# B&R Automation Studio project NAELD004C00R10L518F00 (part 39)

#### Local.var
```iecst
(*2021-08-01*)
(**)
(*Local Action, State & Status*)
VAR
	eAct : eHermesAction := HermesActIdle;
	eStat : eHermesAction := HermesActIdle;
	eMainStatus : eFBStatus := Idle;
	eStatus : eFBStatus := Idle;
	eStatus1 : eFBStatus := Idle;
	eStatus2 : eFBStatus := Idle;
	eStatus3 : eFBStatus := Idle;
	udiStatus : UDINT := 0;
	udiStatus1 : UDINT := 0;
	udiStatus2 : UDINT := 0;
	udiStatus3 : UDINT := 0;
	udiStatus4 : UDINT := 0;
	sStatTxt : STRING[200] := '';
	a_sStatText : ARRAY[0..50] OF STRING[200] := ['Idling','Background Starting Operations','Background Stopping Operations','Deleting Old Log File','Creating Directory','Writing Retain File','Reading Retain File','Saving Configuration',43('')];
END_VAR
(**)
(*Local Alarm*)
VAR
	tyAlmData : tyAlmDat;
	tyAlmData1 : tyAlmDat;
	tyAlmData2 : tyAlmDat;
	tyAlmData3 : tyAlmDat;
	tyAlmData4 : tyAlmDat;
	a_tyAlmText : ARRAY[10000..10199] OF tyAlmTxt := [(sAlmText:='Invalid Ident While Creating Server',sRcyText:='Problem Occurred In The TCP/IP Connection. Check The Connection And Try To Reconnect.'),(sAlmText:='Setting Keep Alive Interval Time Error While Creating Server',sRcyText:='Unable To Establish Connection Between Machine. Check For Setting And Resume Operation.'),(sAlmText:='Setting Keep Alive Idle Time Error While Creating Server',sRcyText:='Unable To Establish Connection Between Machine. Check For Setting And Resume Operation.'),(sAlmText:='Setting Keep Alive Count Error While Creating Server',sRcyText:='Unable To Establish Connection Between Machine. Check For Setting And Resume Operation.'),(sAlmText:='Setting Keep Alive Error While Creating Server',sRcyText:='Unable To Establish Connection Between Machine. Check For Setting And Resume Operation.'),(sAlmText:='Setting Receive Buffer Error While Creating Server',sRcyText:='Unable To Establish Connection Between Machine. Check For Setting And Resume Operation.'),(sAlmText:='Setting Send Buffer Error While Creating Server',sRcyText:='Unable To Establish Connection Between Machine. Check For Setting And Resume Operation.'),(sAlmText:='Setting No Waiting Error While Creating Server',sRcyText:='Unable To Establish Connection Between Machine. Check For Setting And Resume Operation.'),(sAlmText:='TCP Open Port Error While Creating Server',sRcyText:='Problem Occurred In The TCP/IP Connection. Check The Connection And Try To Reconnect.'),(sAlmText:='Closing TCP Error While Creating Server',sRcyText:='Problem Occurred In The TCP/IP Connection. Check The Connection And Try To Reconnect.'),(sAlmText:='Invalid Ident While Listening Client',sRcyText:='There Was A Problem Connecting To The Server. The Server May Not Exist or It is Unavailable At This Time. Check The Connection and Try Again.'),0,(sAlmText:='DS Hermes Connection Lost',sRcyText:='There Was A Problem Connecting To The Server. The Server May Not Exist or It is Unavailable At This Time. Check The Connection and Try Again.'),0,(sAlmText:='Invalid Ident While Receiving Data',sRcyText:='Problem Occurred In The TCP/IP Connection. Check The Connection And Try To Reconnect.'),(sAlmText:='TCP Receive Data Error While Receiving Data',sRcyText:='Problem Occurred In The TCP/IP Connection. Check The Connection And Try To Reconnect.'),(sAlmText:='Receive BoardAvailable While Downstream In Not Connected State',sRcyText:='Receive Illegal Message.'),(sAlmText:='Receive RevokeBoardAvailable While Downstream In Not Connected State',sRcyText:='Receive Illegal Message.'),(sAlmText:='Receive MachineReady While Downstream In Not Connected State',sRcyText:='Receive Illegal Message.'),(sAlmText:='Receive RevokeMachineReady While Downstream In Not Connected State',sRcyText:='Receive Illegal Message.'),(sAlmText:='Receive StartTransport While Downstream In Not Connected State',sRcyText:='Receive Illegal Message.'),(sAlmText:='Receive StopTransport While Downstream In Not Connected State',sRcyText:='Receive Illegal Message.'),(sAlmText:='Receive TransportFinished While Downstream In Not Connected State',sRcyText:='Receive Illegal Message.'),(sAlmText:='Receive BoardForecast While Downstream In Not Connected State',sRcyText:='Receive Illegal Message.'),(sAlmText:='Receive ServiceDescription While Downstream In Service Description State',sRcyText:='Receive Illegal Message.'),(sAlmText:='Receive BoardAvailable While Downstream In Service Description State',sRcyText:='Receive Illegal Message.'),(sAlmText:='Receive RevokeBoardAvailable While Downstream In Service Description State',sRcyText:='Receive Illegal Message.'),(sAlmText:='Receive MachineReady While Downstream In Service Description State',sRcyText:='Receive Illegal Message.'),(sAlmText:='Receive RevokeMachineReady While Downstream In Service Description State',sRcyText:='Receive Illegal Message.'),(sAlmText:='Receive StartTransport While Downstream In Service Description State',sRcyText:='Receive Illegal Message.'),(sAlmText:='Receive StopTransport While Downstream In Service Description State',sRcyText:='Receive Illegal Message.'),(sAlmText:='Receive TransportFinished While Downstream In Service Description State',sRcyText:='Receive Illegal Message.'),(sAlmText:='Receive BoardForecast While Downstream In Service Description State',sRcyText:='Receive Illegal Message.'),(sAlmText:='Receive ServiceDescription While Downstream In Not Available Not Ready State',sRcyText:='Receive Illegal Message.'),(sAlmText:='Receive BoardAvailable While Downstream In Not Available Not Ready State',sRcyText:='Receive Illegal Message.'),(sAlmText:='Receive RevokeBoardAvailable While Downstream In Not Available Not Ready State',sRcyText:='Receive Illegal Message.'),(sAlmText:='Receive RevokeMachineReady While Downstream In Not Available Not Ready State',sRcyText:='Receive Illegal Message.'),(sAlmText:='Receive StartTransport While Downstream In Not Available Not Ready State',sRcyText:='Receive Illegal Message.'),(sAlmText:='Receive StopTransport While Downstream In Not Available Not Ready State',sRcyText:='Receive Illegal Message.'),(sAlmText:='Receive TransportFinished While Downstream In Not Available Not Ready State',sRcyText:='Receive Illegal Message.'),(sAlmText:='Receive BoardForecast While Downstream In Not Available Not Ready State',sRcyText:='Receive Illegal Message.'),(sAlmText:='Receive ServiceDescription While Downstream In Board Available State',sRcyText:='Receive Illegal Message.'),(sAlmText:='Receive BoardAvailable While Downstream In Board Available State',sRcyText:='Receive Illegal Message.'),(sAlmText:='Receive RevokeBoardAvailable While Downstream In Board Available State',sRcyText:='Receive Illegal Message.'),(sAlmText:='Receive RevokeMachineReady While Downstream In Board Available State',sRcyText:='Receive Illegal Message.'),(sAlmText:='Receive StartTransport While Downstream In Board Available State',sRcyText:='Receive Illegal Message.'),(sAlmText:='Receive StopTransport While Downstream In Board Available State',sRcyText:='Receive Illegal Message.'),(sAlmText:='Receive TransportFinished While Downstream In Board Available State',sRcyText:='Receive Illegal Message.'),(sAlmText:='Receive BoardForecast While Downstream In Board Available State',sRcyText:='Receive Illegal Message.'),(sAlmText:='Receive ServiceDescription While Downstream In Machine Ready State',sRcyText:='Receive Illegal Message.'),(sAlmText:='Receive BoardAvailable While Downstream In Machine Ready State',sRcyText:='Receive Illegal Message.'),(sAlmText:='Receive RevokeBoardAvailable While Downstream In Machine Ready State',sRcyText:='Receive Illegal Message.'),(sAlmText:='Receive MachineReady While Downstream In Machine Ready State',sRcyText:='Receive Illegal Message.'),(sAlmText:='Receive StopTransport While Downstream In Machine Ready State',sRcyText:='Receive Illegal Message.'),(sAlmText:='Receive TransportFinished While Downstream In Machine Ready State',sRcyText:='Receive Illegal Message.'),(sAlmText:='Receive BoardForecast While Downstream In Machine Ready State',sRcyText:='Receive Illegal Message.'),(sAlmText:='Receive ServiceDescription While Downstream In Available And Ready State',sRcyText:='Receive Illegal Message.'),(sAlmText:='Receive BoardAvailable While Downstream In Available And Ready State',sRcyText:='Receive Illegal Message.'),(sAlmText:='Receive RevokeBoardAvailable While Downstream In Available And Ready State',sRcyText:='Receive Illegal Message.'),(sAlmText:='Receive MachineReady While Downstream In Available And Ready State',sRcyText:='Receive Illegal Message.'),(sAlmText:='Receive StopTransport While Downstream In Available And Ready State',sRcyText:='Receive Illegal Message.'),(sAlmText:='Receive TransportFinished While Downstream In Available And Ready State',sRcyText:='Receive Illegal Message.'),(sAlmText:='Receive BoardForecast While Downstream In Available And Ready State',sRcyText:='Receive Illegal Message.'),(sAlmText:='Receive ServiceDescription While Downstream In Transporting State',sRcyText:='Receive Illegal Message.'),(sAlmText:='Receive BoardAvailable While Downstream In Transporting State',sRcyText:='Receive Illegal Message.'),(sAlmText:='Receive RevokeBoardAvailable While Downstream In Transporting State',sRcyText:='Receive Illegal Message.'),(sAlmText:='Receive MachineReady While Downstream In Transporting State',sRcyText:='Receive Illegal Message.'),(sAlmText:='Receive RevokeMachineReady While Downstream In Transporting State',sRcyText:='Receive Illegal Message.'),(sAlmText:='Receive StartTransport While Downstream In Transporting State',sRcyText:='Receive Illegal Message.'),(sAlmText:='Receive TransportFinished While Downstream In Transporting State',sRcyText:='Receive Illegal Message.'),(sAlmText:='Receive BoardForecast While Downstream In Transporting State',sRcyText:='Receive Illegal Message.'),(sAlmText:='Receive ServiceDescription While In Transport Finished State',sRcyText:='Receive Illegal Message.'),(sAlmText:='Receive BoardAvailable While In Transport Finished State',sRcyText:='Receive Illegal Message.'),(sAlmText:='Receive RevokeBoardAvailable While In Transport Finished State',sRcyText:='Receive Illegal Message.'),(sAlmText:='Receive MachineReady While In Transport Finished State',sRcyText:='Receive Illegal Message.'),(sAlmText:='Receive RevokeMachineReady While In Transport Finished State',sRcyText:='Receive Illegal Message.'),(sAlmText:='Receive StartTransport While In Transport Finished State',sRcyText:='Receive Illegal Message.'),(sAlmText:='Receive TransportFinished While In Transport Finished State',sRcyText:='Receive Illegal Message.'),(sAlmText:='Receive BoardForecast While In Transport Finished State',sRcyText:='Receive Illegal Message.'),(sAlmText:='Receive ServiceDescription While Downstream In Transport Stopped State',sRcyText:='Receive Illegal Message.'),(sAlmText:='Receive BoardAvailable While Downstream In Transport Stopped State',sRcyText:='Receive Illegal Message.'),(sAlmText:='Receive RevokeBoardAvailable While Downstream In Transport Stopped State',sRcyText:='Receive Illegal Message.'),(sAlmText:='Receive MachineReady While Downstream In Transport Stopped State',sRcyText:='Receive Illegal Message.'),(sAlmText:='Receive RevokeMachineReady While Downstream In Transport Stopped State',sRcyText:='Receive Illegal Message.'),(sAlmText:='Receive StartTransport While Downstream In Transport Stopped State',sRcyText:='Receive Illegal Message.'),(sAlmText:='Receive StopTransport While Downstream In Transport Stopped State',sRcyText:='Receive Illegal Message.'),(sAlmText:='LaneId Mismatch While Checking Service Description',sRcyText:='The LaneId Value Does Not Match. Change The Value And Resend The Value.'),(sAlmText:='MachineId Missing While Checking Service Description',sRcyText:='Missing Input Value For MachineId. Fill Up The Value And Resend.'),(sAlmText:='LandId Out Of Range While Checking Service Description',sRcyText:='LaneId Does Not Fall Within The Expected Range.'),(sAlmText:='LandId Missing While Checking Service Description',sRcyText:='Missing Input Value For LaneId. Fill Up The Value And Resend.'),(sAlmText:='Version Missing While Checking Service Description',sRcyText:='Missing Input Value For Version. Fill Up The Value And Resend.'),(sAlmText:='SupportedFeatures Missing While Checking Service Description',sRcyText:='Missing Input Value For SupportedFeatures. Fill Up The Value And Resend.'),(sAlmText:='NotificationCode Out Of Range While Checking Notification',sRcyText:='NotificationCode Does Not Fall Within The Expected Range.'),(sAlmText:='NotificationCode Missing While Checking Notification',sRcyText:='Missing Input Value For NotificationCode. Fill Up The Value And Resend.'),(sAlmText:='Severity Missing While Checking Notification',sRcyText:='Missing Input Value For Severity. Fill Up The Value And Resend.'),(sAlmText:='Description Missing While Checking Notification',sRcyText:='Missing Input Value For Description. Fill Up The Value And Resend.'),2((0)),(sAlmText:='FailedBoard Missing While Checking Machine Ready',sRcyText:='Missing Input Value For FailedBoard. Fill Up The Value And Resend.'),(sAlmText:='TransferState Missing While Checking Stop Transport',sRcyText:='Missing Input Value For TransferState. Fill Up The Value And Resend.'),(sAlmText:='BoardId Missing While Checking Stop Transport',sRcyText:='Missing Input Value For BoardId. Fill Up The Value And Resend.'),(sAlmText:='BoardId Missing While Checking Start Transport',sRcyText:='Missing Input Value For BoardId. Fill Up The Value And Resend.'),(sAlmText:='Barcode Missing While Checking Query Board Info',sRcyText:='Missing Input Value For BoardId. Fill Up The Value And Resend.'),(0),(sAlmText:='BoardId Mismatch While Checking Start Transport & Stop Transport',sRcyText:='The BoardId Value Does Not Match. Change The Value And Resend The Value.'),(sAlmText:='BoardId Missing While Checking Start Transport & Stop Transport',sRcyText:='Missing Input Value For BoardId. Fill Up The Value And Resend.'),(sAlmText:='Service Description Interchange Time Out',sRcyText:='Timeout Expired Before Operation Completed. Reset And Resume Operation.'),(sAlmText:='Transport Time Out',sRcyText:='Timeout Expired Before Operation Completed. Reset And Resume Operation.'),(sAlmText:='Receive TransportFinished While Downstream In Transport Stopped State',sRcyText:='Receive Illegal Message.'),(sAlmText:='Receive BoardForecast While Downstream In Transport Stopped State',sRcyText:='Receive Illegal Message.'),(sAlmText:='Stop Transport Request To Send From Downstream Hermes',sRcyText:='Sending Illegal Message.'),(sAlmText:='Get Directory Info Error While Deleting Old Log',sRcyText:='An Error Was Encountered While Getting Directory Info. Please Contact Nutek For A Possible Solution.'),(sAlmText:='Directory Read Error While Deleting Old Log',sRcyText:='An Error Was Encountered While Reading Directory. Please Contact Nutek For A Possible Solution.'),(sAlmText:='File Delete Error While Deleting Old Log',sRcyText:='An Error Was Encountered While Trying To Delete File. Please Contact Nutek For A Possible Solution.'),(sAlmText:='File Open Error While Reading Retain File',sRcyText:='An Error Was Encountered While Trying To Open File. Please Contact Nutek For A Possible Solution.'),(sAlmText:='File Read Error While Reading Retain File',sRcyText:='An Error Was Encountered While Trying To Read File. Please Contact Nutek For A Possible Solution.'),(sAlmText:='File Close Error While Reading Retain File',sRcyText:='An Error Was Encountered While Trying To Close File. Please Contact Nutek For A Possible Solution.'),(sAlmText:='File Open Error While Writing Retain File',sRcyText:='An Error Was Encountered While Trying To Open File. Please Contact Nutek For A Possible Solution.'),(sAlmText:='File Create Error While Writing Retain File',sRcyText:='An Error Was Encountered While Trying To Create File. Please Contact Nutek For A Possible Solution.'),(sAlmText:='File Write Error While Writing Retain File',sRcyText:='An Error Was Encountered While Trying To Write File. Please Contact Nutek For A Possible Solution.'),(sAlmText:='File Close Error While Writing Retain File',sRcyText:='An Error Was Encountered While Trying To Close File. Please Contact Nutek For A Possible Solution.'),(sAlmText:='Directory Does Not Exist While Writing Retain File',sRcyText:='The Directory Does Not Exist. Please Contact Nutek For A Possible Solution.'),10((0)),(sAlmText:='Check Alive Time Out',sRcyText:='Timeout Expired Before Operation Completed. Reset And Resume Operation.'),(sAlmText:='Waiting Check Alive Time Out',sRcyText:='Timeout Expired Before Operation Completed. Reset And Resume Operation.'),(sAlmText:='Check Alive Id Mismatch',sRcyText:='The Check Alive Id Value Does Not Match. Change The Value And Resend The Value.'),(sAlmText:='Machine Ready Request To Send From Downstream Hermes',sRcyText:='Sending Illegal Message.'),(sAlmText:='Revoke Machine Ready Request To Send From Downstream Hermes',sRcyText:='Sending Illegal Message.'),(sAlmText:='Start Transport Request To Send From Downstream Hermes',sRcyText:='Sending Illegal Message.'),(sAlmText:='Set Configuration Request To Send From Downstream Hermes',sRcyText:='Sending Illegal Message.'),(sAlmText:='Get Configuration Request To Send From Downstream Hermes',sRcyText:='Sending Illegal Message.'),(sAlmText:='Current Configuration Request To Send From Downstream Hermes',sRcyText:='Sending Illegal Message.'),(sAlmText:='Board Forecast Request To Send From Downstream Hermes',sRcyText:='Sending Illegal Message.'),(sAlmText:='Query Board Info Request To Send From Downstream Hermes',sRcyText:='Sending Illegal Message.'),(sAlmText:='Invalid Ident While Sending Data',sRcyText:='Invalid Ident Value.'),(sAlmText:='TCP Retry Send Data Error While Sending Data',sRcyText:='Problem Occurred In The TCP/IP Connection. Check The Connection And Try To Reconnect.'),(sAlmText:='TCP Send Data Error',sRcyText:='Problem Occurred In The TCP/IP Connection. Check The Connection And Try To Reconnect.'),(sAlmText:='Invalid Ident While Closing TCP',sRcyText:='Invalid Ident Value.'),(sAlmText:='Closing TCP Error',sRcyText:='Problem Occurred In The TCP/IP Connection. Check The Connection And Try To Reconnect.'),(sAlmText:='File Open Error While Writing Log',sRcyText:='An Error Was Encountered While Trying To Open File. Please Contact Nutek For A Possible Solution.'),(sAlmText:='File Create Error While Writing Log',sRcyText:='An Error Was Encountered While Trying To Create File. Please Contact Nutek For A Possible Solution.'),(sAlmText:='Get File Info Error While Writing Log',sRcyText:='An Error Was Encountered While Getting File Info. Please Contact Nutek For A Possible Solution.'),(sAlmText:='File Write Error While Writing Log',sRcyText:='An Error Was Encountered While Trying To Write File. Please Contact Nutek For A Possible Solution.'),(sAlmText:='File Close Error While Writing Log',sRcyText:='An Error Was Encountered While Trying To Close File. Please Contact Nutek For A Possible Solution.'),(sAlmText:='Directory Does Not Exist While Writing Log',sRcyText:='The Directory Does Not Exist.Please Contact Nutek For A Possible Solution.'),(sAlmText:='Invalid Ident While Closing TCP',sRcyText:='Invalid Ident Value.'),(sAlmText:='Closing TCP Error',sRcyText:='Problem Occurred In The TCP/IP Connection. Check The Connection And Try To Reconnect.'),0,(sAlmText:='Board Jam At Sensor After Transfer Interrupted',sRcyText:='Pull Back Board From Downstream Machine'),0,(sAlmText:='Send Board Info Request To Send From Downstream Hermes',sRcyText:='Sending Illegal Message.'),(sAlmText:='Query Work Order Info Request To Send From Downstream Hermes',sRcyText:='Sending Illegal Message.'),(sAlmText:='Send Work Order Info Request To Send From Downstream Hermes',sRcyText:='Sending Illegal Message.'),(sAlmText:='Board Arrived Request To Send From Downstream Hermes',sRcyText:='Sending Illegal Message.'),(sAlmText:='Board departed Request To Send From Downstream Hermes',sRcyText:='Sending Illegal Message.'),(sAlmText:='Forecast Id Mismatch While Checking BoardForecast & Machine Ready',sRcyText:='The ForecastId Value Does Not Match. Change The Value And Resend The Value.'),(sAlmText:='Product Type Id Mismatch While Checking BoardForecast & Machine Ready',sRcyText:='The ProductTypetId Value Does Not Match. Change The Value And Resend The Value.'),(sAlmText:='Width Mismatch While Checking BoardForecast & Machine Ready',sRcyText:='The Width Value Does Not Match. Change The Value And Resend The Value.'),(sAlmText:='Query Top Barcode and Bottom Barcode found from different Recipes',sRcyText:='Please Check or Scan Again the PCB Barcode'),32(0)];
END_VAR
(**)
(*Local Output*)
VAR
	bConnected : BOOL;
	bHandshakeDone : BOOL;
	bSendOk : BOOL;
	bSearchTop : BOOL;
	bSearchBottom : BOOL;
	bFoundIndex : BOOL;
	bFoundTop : BOOL;
	bFoundBottom : BOOL;
	bFoundNothing : BOOL;
	bNewChangeOver : BOOL;
	bSendBFId : BOOL;
	bRstSendBFId : BOOL;
	bUSRdy : BOOL;
	bDSRdy : BOOL;
	bUSGdRdy : BOOL;
	bDSGdRdy : BOOL;
	bTransporting : BOOL;
	bStopTransport : BOOL;
	sInternalSnd : STRING[65535];
	bTransportFinishedSnd : BOOL;
	tyBoardDepartedInfo : tyHermesBoardAvailable;
END_VAR
(**)
(*Local Input*)
VAR
	udiRstErr : UDINT := 0;
	bPrep : BOOL := TRUE;
	bEn : BOOL := TRUE;
	bDis : BOOL := FALSE;
	tyParam : tyHermesDSParam;
	sIPAddr : STRING[15] := '192.168.0.100';
	a_usiMacAddr : ARRAY[0..5] OF USINT := [6(0)];
	tyDTStructure : DTStructure := (year:=2020,month:=11,day:=11,wday:=05,hour:=21,minute:=28,second:=30,millisec:=123,microsec:=456);
	dtCurrDT : DATE_AND_TIME := DT#2019-02-23-12:30:50;
	bRdySnd : BOOL := FALSE;
	bSndCompl : BOOL := FALSE;
	bSndInCompl : BOOL := FALSE;
	bSndNotStart : BOOL := FALSE;
	bFirstZoneEndSen : BOOL;
	bBAWidthEn : BOOL := TRUE; (*Board Available Check Width*)
	bBASltEn : BOOL := TRUE; (*Board Available Check Slot*)
	bBFWidthEn : BOOL := TRUE; (*Board Forecast Check Width*)
	bBFSltEn : BOOL := FALSE; (*Board Forecst Check Slot*)
	sForecastId : {REDUND_UNREPLICABLE} STRING[80] := '';
	sBoardId : STRING[36] := '';
	sMcId : STRING[80] := '';
	sInterfaceId : STRING[80] := '';
	sVersion : STRING[7] := '1.3';
	eFailedBoard : eHermesFailedBoard := HermesUnknownBoard;
	sRecipeNm : STRING[254] := '';
	eFlippedBoard : eHermesFlippedBoard := HermesFlippedBoardUnknownSide;
	sTopBarcode : STRING[254] := '';
	sBottomBarcode : STRING[254] := '';
	rLength : REAL := 0;
	rThickness : REAL := 0;
	rConveyorSpeed : REAL := 0;
	rTopClearanceHeight : REAL := 0;
	rBottomClearanceHeight : REAL := 0;
	rWeight : REAL := 0;
	sWorkOrderId : STRING[80] := '';
	sBatchId : STRING[80] := '';
	diWidthInUM : DINT := 0;
	diMinSltValue : DINT := 0;
	diMaxSltValue : DINT := 0;
	diPitch : DINT := 0;
	diTtlSlt : DINT := 0;
	diSltToSltInUM : DINT := 0;
	udiSndBffrSize : UDINT := 65536;
	udiRcvBffrSize : UDINT := 65536;
	udiAliveIdleTimeInSec : UDINT := 5;
	tConnTimeOut : TIME := T#30s;
	diTransferInTO : DINT := 30000;
	a_tyXMLTableDataBrdAvl : ARRAY[0..200] OF tyXMLTableDat;
	iXMLTableDataBrdAvlTtlIdx : INT := 0;
	bNewBrdAvl1 : BOOL := FALSE;
	bNewBrdAvl2 : BOOL := FALSE;
	bOpsRun : BOOL := FALSE;
	bInterruptSen : BOOL := FALSE;
	udiFileKeepDay : UDINT := 30;
	sRetainFileName : STRING[80] := 'BoardData.dat';
	sProgNm : STRING[15] := 'DSHermes';
	bNtSettingsLoadDone : BOOL := TRUE;
	bRmtPrep : BOOL := FALSE;
	bRmtEn : BOOL := FALSE;
	bSvyPrep : BOOL := FALSE;
	bSvyEn : BOOL := FALSE;
	bAllZonesEmpty : BOOL := FALSE;
	bFirstZoneHaveBoard : BOOL := FALSE;
	bInternalUse : BOOL;
	sInternalRcv : STRING[65535];
	rMachineCycleTime : REAL := 6000;
	rAutoWidthCycleTime : REAL := 30000;
	tyHermesCurrConfiguration : tyHermesConfiguration;
	tyBoardInfoData : tyHermesSendBoardInfo;
	tyUSBoardArrivedData : tyHermesBoardAvailable;
	bUSHermesStopTransport : BOOL;
	bRcvBoardInfo : BOOL;
	bUSHermesTransporting : BOOL;
	bOpsGConv1HvBrd : BOOL;
END_VAR
(**)
(*Local*)
VAR
	bRstErr : BOOL;
	udiRstErrOld : UDINT;
	bInitDone : BOOL;
	bInitialDone : BOOL;
	bRun : BOOL;
	bStop : BOOL;
	bRstConnection : BOOL;
	bRstState : BOOL;
	udiSvrIdent : UDINT;
	udiClntIdent : UDINT;
	udiClntIdentExtra : UDINT;
	udiXMLTableWriteIdx : UDINT;
	udiMsgSendBffr : UDINT;
	udiSndMsgLen : UDINT;
	sSnd : STRING[65535];
	sRcv : STRING[65535];
	a_tyXMLTableDataRcv : ARRAY[0..200] OF tyXMLTableDat;
	a_tyXMLTableDataSnd : ARRAY[0..200] OF tyXMLTableDat;
	a_eMsgSend : ARRAY[0..50] OF eHermesMsgType;
	tyMsgTypeRcv : tyHermesMsgType;
	tyCheckAliveSnd : tyHermesCheckAlive;
	tyCheckAlivePingSnd : tyHermesCheckAlive;
	tyCheckAlivePongSnd : tyHermesCheckAlive;
	tyCheckAliveRcv : tyHermesCheckAlive;
	tyCheckAlivePingRcv : tyHermesCheckAlive;
	tyCheckAlivePongRcv : tyHermesCheckAlive;
	tyServiceDescriptionSnd : tyHermesServiceDescription;
	tyServiceDescriptionRcv : tyHermesServiceDescription;
	tyNotificationSnd : tyHermesNotification;
	tyNotificationRcv : tyHermesNotification;
	tyBoardAvailableRcv : tyHermesBoardAvailable;
	tyBoardAvailableSnd : tyHermesBoardAvailable;
	a_tyBoardDepartedInfo : ARRAY[0..49] OF tyHermesBoardAvailable;
	tyMachineReady : tyHermesMachineReady;
	tyStartTransport : tyHermesStartTransport;
	tyStopTransport : tyHermesStopTransport;
	tyTransportFinished : tyHermesTransportFinished;
	tySetConfiguration : tyHermesSetConfiguration;
	tyCurrentConfiguration : tyHermesCurrentConfiguration;
	tyBoardForecastRcv : tyHermesBoardForecast;
	tyBoardForecastSnd : tyHermesBoardForecast;
	tyQueryBoardInfo : tyHermesQueryBoardInfo;
	tySendBoardInfo : tyHermesSendBoardInfo;
	fbCreateSvr : fbTCPCreateSvr;
	fbListen : fbTCPListen;
	fbRcv : fbTCPRcv;
	fbSend : fbTCPSnd;
	fbCloseSvr : fbTCPClose;
	fbCloseClnt : fbTCPClose;
	fbParseXMLTable : fbHermesParseXMLTable;
	fbParseBrdAvlExternal : fbHermesParseXMLTable;
	fbCheckAlive : fbHermesCheckAlive;
	fbCheckAliveSendPing : fbHermesCheckAliveSendPing;
	fbCheckAliveRcvPing : fbHermesCheckAliveRcvPing;
	fbSequenceDS : fbHermesSequenceDS;
	fbSequenceTO : fbHermesSequenceTO;
	eStatOld : eHermesAction := HermesActIdle;
	tyParamOld : tyHermesDSParam;
	bFeatureBoardForecast : BOOL;
	bNewProduct : USINT;
	bNewWidth : BOOL;
	bSiemensNewProduct : BOOL;
	bTest888 : BOOL;
	idxBoardForecastId : INT := 0;
	idxBoardForecastNoId : INT := 0;
END_VAR
VAR RETAIN
	udiBAIndex : UDINT := 0;
END_VAR
VAR
	i : UDINT := 0;
	j : UDINT := 0;
	jj : UDINT := 0;
	udiTopTargetAddress : UDINT := 0;
	udiBottomTargetAddress : UDINT := 0;
	udiSizeOfAddress : UDINT := 0;
	udiTargetAddress : UDINT := 0;
	udiSizeAddress : UDINT := 0;
	udiFoundAddressTop : UDINT := 0;
	udiFoundRecipeTop : UDINT := 0;
	udiFoundRecipeFinal : UDINT := 0;
	udiFoundAddressBottom : UDINT := 0;
	udiFoundRecipeBottom : UDINT := 0;
	sSearchTop : STRING[254] := '';
	sSearchBottom : STRING[254] := '';
	udiLogCntr : UDINT := 1;
	udiWriteLogCntr : UDINT := 1;
	a_sLogList : ARRAY[1..10] OF STRING[65535];
	sDT : STRING[80];
	dtCurrDTTemp : DATE_AND_TIME;
	fbFileAppend1 : fbFileFullAppend;
	fbFileOldDel1 : fbFileOldDel;
	fbFileRead1 : fbFileFullRead;
	fbFileWrite1 : fbFileFullWrite;
	fbSendTm : TON;
	bFileNotFound : BOOL;
	udiRetainDataAddr : UDINT;
	udiRetainDataLen : UDINT;
	iWriteLogStep : INT := 0;
	fbDeleteLogTmr : TON := (PT:=T#24h);
	fbDlyTmr : TON := (PT:=T#5s);
	fbSendBFRstTmr : TON := (PT:=T#10s);
	udiModuleNum : UDINT := 3351;
	bBFAccNewWidth : ARRAY[1..3] OF BOOL := [3(FALSE)];
END_VAR
```

#### Act_Alarm.st
```iecst
(** 2021-08-01 **)
ACTION Act_Alarm:

	//Error
	IF EDGEPOS(eStatus = Error) THEN

		tyAlmData.sProgNm		:= p_sProgNm;
		tyAlmData.udiCode		:= udiStatus;
		tyAlmData.eSeverity		:= AlmSeverityError;
		tyAlmData.udiRunTime	:= tyAlmData.udiRunTime + 1;
		tyAlmData.bAlm			:= TRUE;
		tyAlmData.udiModuleNum  := udiModuleNum;
		g_sDSHermesAProgNm		:= p_sProgNm;
		//Get Error Message
		IF tyAlmData.udiCode < 10000 OR tyAlmData.udiCode > 10199 THEN
			tyAlmData.sAlmMsg	:= 'Unknown';
			tyAlmData.sRcyMsg	:= 'Unknown';
		ELSE
			tyAlmData.sAlmMsg	:= a_tyAlmText[tyAlmData.udiCode].sAlmText;
			tyAlmData.sRcyMsg	:= a_tyAlmText[tyAlmData.udiCode].sRcyText;
		END_IF

		sStatTxt	:= tyAlmData.sAlmMsg;

	ELSIF bRstErr AND (tyAlmData.udiCode <> 0) THEN

		tyAlmData.udiCode	:= 0;
		tyAlmData.eSeverity	:= AlmSeverityNA;
		tyAlmData.sAlmMsg	:= '';
		tyAlmData.sRcyMsg	:= '';
		tyAlmData.bAlm			:= FALSE;
		sStatTxt	:= a_sStatText[eStat];

	END_IF

END_ACTION
```

#### Act_Alarm1.st
```iecst
(** 2021-08-01 **)
ACTION Act_Alarm1: //General

	//Error
	IF EDGEPOS(eStatus1 = Error) THEN

		tyAlmData1.sProgNm		:= p_sProgNm;
		tyAlmData1.udiCode		:= udiStatus1;
		tyAlmData1.eSeverity	:= AlmSeverityError;
		tyAlmData1.udiRunTime	:= tyAlmData1.udiRunTime + 1;
		tyAlmData1.bAlm			:= TRUE;
		tyAlmData1.udiModuleNum  := udiModuleNum;
		g_sDSHermesAProgNm		:= p_sProgNm;

		//Get Error Message
		IF tyAlmData1.udiCode < 10000 OR tyAlmData1.udiCode > 10199 THEN
			tyAlmData1.sAlmMsg	:= 'Unknown';
			tyAlmData1.sRcyMsg	:= 'Unknown';
		ELSE
			tyAlmData1.sAlmMsg	:= a_tyAlmText[tyAlmData1.udiCode].sAlmText;
			tyAlmData1.sRcyMsg	:= a_tyAlmText[tyAlmData1.udiCode].sRcyText;
		END_IF

		sStatTxt	:= tyAlmData1.sAlmMsg;

	ELSIF bRstErr AND (tyAlmData1.udiCode <> 0) THEN

		tyAlmData1.udiCode		:= 0;
		tyAlmData1.eSeverity	:= AlmSeverityNA;
		tyAlmData1.sAlmMsg		:= '';
		tyAlmData1.sRcyMsg		:= '';
		tyAlmData1.bAlm			:= FALSE;
		sStatTxt	:= a_sStatText[eStat];

	END_IF

END_ACTION
```

#### Act_Alarm2.st
```iecst
(** 2019-03-25 **)
ACTION Act_Alarm2:

	//Error
	IF EDGEPOS(eStatus2 = Error) THEN

		tyAlmData2.sProgNm		:= p_sProgNm;
		tyAlmData2.udiCode		:= udiStatus2;
		tyAlmData2.eSeverity	:= AlmSeverityError;
		tyAlmData2.udiRunTime	:= tyAlmData2.udiRunTime + 1;
		tyAlmData2.bAlm			:= TRUE;
		tyAlmData2.udiModuleNum  := udiModuleNum;
		g_sDSHermesAProgNm		:= p_sProgNm;
		//Get Error Message
		IF tyAlmData2.udiCode < 10000 OR tyAlmData2.udiCode > 10199 THEN
			tyAlmData2.sAlmMsg	:= 'Unknown';
			tyAlmData2.sRcyMsg	:= 'Unknown';
		ELSE
			tyAlmData2.sAlmMsg	:= a_tyAlmText[tyAlmData2.udiCode].sAlmText;
			tyAlmData2.sRcyMsg	:= a_tyAlmText[tyAlmData2.udiCode].sRcyText;
		END_IF

		sStatTxt	:= tyAlmData2.sAlmMsg;

	ELSIF bRstErr AND (tyAlmData2.udiCode <> 0) THEN

		tyAlmData2.udiCode		:= 0;
		tyAlmData2.eSeverity	:= AlmSeverityNA;
		tyAlmData2.sAlmMsg		:= '';
		tyAlmData2.sRcyMsg		:= '';
		tyAlmData2.bAlm			:= FALSE;
		sStatTxt	:= a_sStatText[eStat];

	END_IF

END_ACTION
```

#### Act_Alarm3.st
```iecst
(** 2021-08-01 **)
ACTION Act_Alarm3: //fbFileAppend1 Error

	//Error
	IF EDGEPOS(eStatus3 = Error) THEN

		tyAlmData3.sProgNm		:= p_sProgNm;
		tyAlmData3.udiCode		:= udiStatus3;
		tyAlmData3.eSeverity	:= AlmSeverityError;
		tyAlmData3.udiRunTime	:= tyAlmData3.udiRunTime + 1;
		tyAlmData3.bAlm			:= TRUE;
		tyAlmData3.udiModuleNum  := udiModuleNum;
		g_sDSHermesAProgNm		:= p_sProgNm;
		//Get Error Message
		IF tyAlmData3.udiCode < 10000 OR tyAlmData3.udiCode > 10199 THEN
			tyAlmData3.sAlmMsg	:= 'Unknown';
			tyAlmData3.sRcyMsg	:= 'Unknown';
		ELSE
			tyAlmData3.sAlmMsg	:= a_tyAlmText[tyAlmData3.udiCode].sAlmText;
			tyAlmData3.sRcyMsg	:= a_tyAlmText[tyAlmData3.udiCode].sRcyText;
		END_IF

		sStatTxt	:= tyAlmData3.sAlmMsg;

	ELSIF bRstErr AND (tyAlmData3.udiCode <> 0) THEN

		tyAlmData3.udiCode		:= 0;
		tyAlmData3.eSeverity	:= AlmSeverityNA;
		tyAlmData3.sAlmMsg		:= '';
		tyAlmData3.sRcyMsg		:= '';
		tyAlmData3.bAlm			:= FALSE;
		sStatTxt	:= a_sStatText[eStat];

	END_IF

END_ACTION
```

#### Act_Alarm4.st
```iecst
(** 2021-08-01 **)
ACTION Act_Alarm4: //Not Connected Warning

	//Warning
	IF ((bConnected = FALSE) AND (p_eLinkMcParamDSCommMod= McSetCommModHermes)) THEN

		tyAlmData4.sProgNm		:= p_sProgNm;
		tyAlmData4.udiCode		:= udiStatus4;
		tyAlmData4.eSeverity	:= AlmSeverityWarning;
		tyAlmData4.udiRunTime	:= tyAlmData4.udiRunTime + 1;
		tyAlmData4.bWarning			:= TRUE;
		tyAlmData4.udiModuleNum  := udiModuleNum;
		g_sDSHermesAProgNm		:= p_sProgNm;
		//Get Error Message
		IF tyAlmData4.udiCode < 10000 OR tyAlmData4.udiCode > 10199 THEN
			tyAlmData4.sAlmMsg	:= 'Unknown';
			tyAlmData4.sRcyMsg	:= 'Unknown';
		ELSE
			tyAlmData4.sAlmMsg	:= a_tyAlmText[tyAlmData4.udiCode].sAlmText;
			tyAlmData4.sRcyMsg	:= a_tyAlmText[tyAlmData4.udiCode].sRcyText;
		END_IF

		sStatTxt	:= tyAlmData4.sAlmMsg;

	ELSIF (bConnected AND (tyAlmData4.udiCode <> 0)) OR (p_eLinkMcParamDSCommMod= McSetCommModSMEMA) THEN

		tyAlmData4.udiCode		:= 0;
		tyAlmData4.eSeverity	:= AlmSeverityNA;
		tyAlmData4.sAlmMsg		:= '';
		tyAlmData4.sRcyMsg		:= '';
		tyAlmData4.bWarning			:= FALSE;
		sStatTxt	:= a_sStatText[eStat];

	END_IF

END_ACTION
```

#### Act_Background.st
```iecst
(** 2021-08-01 **)
ACTION Act_Background:

	IF bRun = TRUE THEN
		IF udiSvrIdent = 0 THEN
			IF p_bInternalUse = FALSE THEN
				Act_Background_TCPCreateSvr;

				tyParamOld	:= p_tyParam;
			ELSE
				udiSvrIdent	:= 1;
			END_IF

		ELSE
			IF bRstConnection = FALSE THEN

				Act_Background_ChgConfig;

				IF udiClntIdent = 0 THEN
					IF p_bInternalUse = FALSE THEN
						Act_Background_TCPListen;
					ELSE
						udiClntIdent	:= 1;
					END_IF

				ELSE
					Act_Background_TCPRcv;

					Act_Background_NotificationRcv;

					Act_Background_IllegalMsg;
					Act_Background_ChkParamRcv;
					Act_Background_CmpParamRcv;

					IF bHandshakeDone = TRUE THEN
						IF (p_tyParam.tSndAlive <> T#0s) AND (p_tyParam.tRcvAlive <> T#0s) THEN
							IF tyServiceDescriptionRcv.tyData.tySupportedFeatures.bFeatureCheckAliveResponse = TRUE AND p_tyParam.bFeatureCheckAliveResponse = TRUE THEN
								Act_Background_ChkAliveSendPing;
								Act_Background_ChkAliveRcvPing;
							ELSE
								Act_Background_ChkAlive;
							END_IF
						ELSE
							fbCheckAlive(bEn := FALSE);
							fbCheckAliveSendPing(bEn := FALSE);
							fbCheckAliveRcvPing(bEn := FALSE);
						END_IF
					END_IF

					Act_Background_Sequence;
					Act_Background_SequenceTO;
					Act_Background_Err;

					IF tyServiceDescriptionRcv.tyAvl.tySupportedFeatures.bFeatureQueryBoardInfo = TRUE AND p_tyParam.bFeatureSendBoardInfo AND bHandshakeDone THEN
						Act_Background_SendBoardInfo;
					END_IF

					Act_Background_TCPSend;
					Act_Background_Log;

				END_IF

			ELSE
				IF udiClntIdent <> 0 THEN
					Act_Background_TCPCloseClnt;
				ELSE
					IF udiSvrIdent <> 0 THEN
						Act_Background_TCPCloseSvr;
					END_IF
				END_IF

			END_IF

			//Second Client Connected
			IF udiClntIdentExtra = 0 THEN

			ELSE

			END_IF

		END_IF

		Act_Background_Stop;

	END_IF

	IF EDGENEG(bRun) OR EDGENEG(udiSvrIdent = 0) THEN
		//Reset
		fbCreateSvr(bEn := FALSE);
	END_IF

	IF EDGENEG(bRun) OR EDGENEG(udiClntIdent = 0) THEN
		//Reset
		fbListen(bEn := FALSE);

		bConnected	:= bRun;
	END_IF

	IF EDGENEG(bRun) OR EDGENEG(udiSvrIdent <> 0) OR EDGENEG(udiClntIdent <> 0) THEN
		fbRcv(bEn := FALSE);
		fbSequenceDS(bEn := FALSE);
		fbSequenceTO(bEn := FALSE);
		fbCheckAlive(bEn := FALSE);
		fbCheckAliveSendPing(bEn := FALSE);
		fbCheckAliveRcvPing(bEn := FALSE);
		fbSend(bEn := FALSE);

		fbFileAppend1(bEn := FALSE);
		iWriteLogStep	:= 0;

		bConnected		:= FALSE;
		bHandshakeDone	:= FALSE;
		bRstState		:= FALSE;
		bUSRdy			:= FALSE;
		bDSRdy			:= FALSE;
		bTransporting	:= FALSE;
		bStopTransport	:= FALSE;

		memset(ADR(tyMsgTypeRcv) , 0 , SIZEOF(tyMsgTypeRcv));
		memset(ADR(a_eMsgSend) , 0 , SIZEOF(a_eMsgSend));
		udiMsgSendBffr	:= 0;
	END_IF

	IF EDGENEG(bRun) OR EDGENEG(udiSvrIdent <> 0) THEN
		bRstConnection	:= FALSE;
		fbCloseSvr(bEn := FALSE);
	END_IF

	IF EDGENEG(bRun) OR EDGENEG(udiClntIdent <> 0) THEN
		fbCloseClnt(bEn := FALSE);
	END_IF

	//Reset Error
	IF (eStatus1 = Error) AND bRstErr THEN
		eStatus1	:= Idle;
		udiStatus1	:= 0;

		fbCreateSvr(bEn := FALSE);
		fbListen(bEn := FALSE);
		fbRcv(bEn := FALSE);
		fbSequenceDS(bEn := FALSE);
		fbSend(bEn := FALSE);
		fbCloseSvr(bEn := FALSE);
		fbCloseClnt(bEn := FALSE);
		fbCheckAlive(bEn := FALSE);
		fbCheckAliveSendPing(bEn := FALSE);
		fbCheckAliveRcvPing(bEn := FALSE);
		fbSequenceTO(bEn := FALSE);

		fbFileAppend1(bEn := FALSE);
		iWriteLogStep	:= 0;

		bConnected		:= FALSE;
		bHandshakeDone	:= FALSE;
		bRstConnection	:= FALSE;
		bRstState		:= FALSE;
		bUSRdy			:= FALSE;
		bDSRdy			:= FALSE;
		bTransporting	:= FALSE;
		bStopTransport	:= FALSE;

		memset(ADR(tyMsgTypeRcv) , 0 , SIZEOF(tyMsgTypeRcv));
		memset(ADR(a_eMsgSend) , 0 , SIZEOF(a_eMsgSend));
		udiMsgSendBffr	:= 0;
	END_IF

	IF (eStatus2 = Error) AND bRstErr THEN
		eStatus2	:= Idle;
		udiStatus2	:= 0;

		fbSequenceTO(bEn := FALSE);

	END_IF

	IF (eStatus3 = Error) AND bRstErr THEN
		eStatus3	:= Idle;
		udiStatus3	:= 0;

		fbFileAppend1(bEn := FALSE);
		iWriteLogStep	:= 0;
	END_IF

END_ACTION
```

#### Act_Background_ChkAlive.st
```iecst
(** 2021-08-01 **)
ACTION Act_Background_ChkAlive:

	IF eStatus1 <> Error THEN

		//Standard Check Alive (Without Ping & Pong)
		fbCheckAlive.bDataRcv		:= tyMsgTypeRcv.bCheckAlive OR tyMsgTypeRcv.bMachineReady OR tyMsgTypeRcv.bRevokeMachineReady OR tyMsgTypeRcv.bStartTransport OR tyMsgTypeRcv.bStopTransport OR tyMsgTypeRcv.bQueryBoardInfo;
		fbCheckAlive.tSendTm		:= p_tyParam.tSndAlive;
		fbCheckAlive.tRcvTimeOut	:= p_tyParam.tRcvAlive;
		fbCheckAlive(bEn := TRUE);

		IF fbCheckAlive.udiStatus > 0 AND fbCheckAlive.udiStatus < 65534 THEN
			eStatus1	:= Error;

			IF fbCheckAlive.udiStatus = 2767 THEN
				udiStatus1	:= 10132;	//Check Alive Time Out
			ELSE
				udiStatus1	:= fbCheckAlive.udiStatus;
			END_IF

			fHermesAddOneMsgSend(ADR(a_eMsgSend) , ADR(udiMsgSendBffr) , HermesMsgTypeNotification);

			tyNotificationSnd.tyAvl.bSeverity			:= TRUE;
			tyNotificationSnd.tyAvl.bNotificationCode	:= TRUE;
			tyNotificationSnd.tyAvl.bDescription		:= TRUE;
			tyNotificationSnd.tyData.eSeverity			:= HermesSeverityFatalError;
			tyNotificationSnd.tyData.iNotificationCode	:= UDINT_TO_INT(udiStatus1);
			tyNotificationSnd.tyData.sDescription		:= a_tyAlmText[udiStatus1].sAlmText;

		ELSE
			IF EDGEPOS(fbCheckAlive.bDataSend) THEN
				fHermesAddOneMsgSend(ADR(a_eMsgSend) , ADR(udiMsgSendBffr) , HermesMsgTypeCheckAlive);
				tyCheckAliveSnd	:= fbCheckAlive.tyDataSend;
			END_IF

		END_IF

		tyMsgTypeRcv.bCheckAlive	:= FALSE;	//Reset Check Alive

	END_IF

END_ACTION
```

#### Act_Background_ChkParamRcv.st
```iecst
(** 2021-08-01 **)
ACTION Act_Background_ChkParamRcv:

	IF eStatus2 <> Error THEN

		//Check Parameter Receive
		IF tyMsgTypeRcv.bServiceDescription = TRUE THEN
			udiStatus2	:= fHermesChkParamSD(tyServiceDescriptionRcv , p_tyParam.iLaneID);

			IF udiStatus2 = 2731 THEN
				udiStatus2	:= 0;
			END_IF

			IF udiStatus2 <> 0 THEN
				eStatus2	:= Error;

				IF udiStatus2 = 2726 THEN
					udiStatus2	:= 10086;	//LaneId Mismatch While Checking Service Description
				ELSIF udiStatus2 = 2727 THEN
					udiStatus2	:= 10087;	//MachineId Missing While Checking Service Description
				ELSIF udiStatus2 = 2728 THEN
					udiStatus2	:= 10088;	//LandId Out Of Range While Checking Service Description
				ELSIF udiStatus2 = 2729 THEN
					udiStatus2	:= 10089;	//LandId Missing While Checking Service Description
				ELSIF udiStatus2 = 2730 THEN
					udiStatus2	:= 10090;	//Version Missing While Checking Service Description
				ELSIF udiStatus2 = 2731 THEN
					udiStatus2	:= 10091;	//SupportedFeatures Missing While Checking Service Description
				END_IF

				fHermesAddOneMsgSend(ADR(a_eMsgSend) , ADR(udiMsgSendBffr) , HermesMsgTypeNotification);

				tyNotificationSnd.tyAvl.bSeverity			:= TRUE;
				tyNotificationSnd.tyAvl.bNotificationCode	:= TRUE;
				tyNotificationSnd.tyAvl.bDescription		:= TRUE;
				tyNotificationSnd.tyData.eSeverity			:= HermesSeverityFatalError;
				tyNotificationSnd.tyData.iNotificationCode	:= UDINT_TO_INT(udiStatus2);
				tyNotificationSnd.tyData.sDescription		:= a_tyAlmText[udiStatus2].sAlmText;

			END_IF
		END_IF

		IF tyMsgTypeRcv.bNotification = TRUE THEN
			udiStatus2	:= fHermesChkParamN(tyNotificationRcv);

			IF udiStatus2 <> 0 THEN
				eStatus2	:= Error;

				IF udiStatus2 = 2732 THEN
					udiStatus2	:= 10092;	//NotificationCode Out Of Range While Checking Notification
				ELSIF udiStatus2 = 2733 THEN
					udiStatus2	:= 10093;	//NotificationCode Missing While Checking Notification
				ELSIF udiStatus2 = 2734 THEN
					udiStatus2	:= 10094;	//Severity Missing While Checking Notification
				ELSIF udiStatus2 = 2735 THEN
					udiStatus2	:= 10095;	//Description Missing While Checking Notification
				END_IF

				fHermesAddOneMsgSend(ADR(a_eMsgSend) , ADR(udiMsgSendBffr) , HermesMsgTypeNotification);

				tyNotificationSnd.tyAvl.bSeverity			:= TRUE;
				tyNotificationSnd.tyAvl.bNotificationCode	:= TRUE;
				tyNotificationSnd.tyAvl.bDescription		:= TRUE;
				tyNotificationSnd.tyData.eSeverity			:= HermesSeverityFatalError;
				tyNotificationSnd.tyData.iNotificationCode	:= UDINT_TO_INT(udiStatus2);
				tyNotificationSnd.tyData.sDescription		:= a_tyAlmText[udiStatus2].sAlmText;

			END_IF
		END_IF

		IF tyMsgTypeRcv.bMachineReady = TRUE THEN
			udiStatus2	:= fHermesChkParamMR(tyMachineReady);

			IF udiStatus2 <> 0 THEN
				eStatus2	:= Error;

				IF udiStatus2 = 2740 THEN
					udiStatus2	:= 10098;	//FailedBoard Missing While Checking Machine Ready
				END_IF

				fHermesAddOneMsgSend(ADR(a_eMsgSend) , ADR(udiMsgSendBffr) , HermesMsgTypeNotification);

				tyNotificationSnd.tyAvl.bSeverity			:= TRUE;
				tyNotificationSnd.tyAvl.bNotificationCode	:= TRUE;
				tyNotificationSnd.tyAvl.bDescription		:= TRUE;
				tyNotificationSnd.tyData.eSeverity			:= HermesSeverityError;
				tyNotificationSnd.tyData.iNotificationCode	:= UDINT_TO_INT(udiStatus2);
				tyNotificationSnd.tyData.sDescription		:= a_tyAlmText[udiStatus2].sAlmText;

			END_IF
		END_IF

		IF tyMsgTypeRcv.bStartTransport = TRUE THEN
			udiStatus2	:= fHermesChkParamSAT(tyStartTransport);

			IF udiStatus2 <> 0 THEN
				eStatus2	:= Error;

				IF udiStatus2 = 2745 THEN
					udiStatus2	:= 10101;	//BoardId Missing While Checking Start Transport
				END_IF

				fHermesAddOneMsgSend(ADR(a_eMsgSend) , ADR(udiMsgSendBffr) , HermesMsgTypeNotification);

				tyNotificationSnd.tyAvl.bSeverity			:= TRUE;
				tyNotificationSnd.tyAvl.bNotificationCode	:= TRUE;
				tyNotificationSnd.tyAvl.bDescription		:= TRUE;
				tyNotificationSnd.tyData.eSeverity			:= HermesSeverityError;
				tyNotificationSnd.tyData.iNotificationCode	:= UDINT_TO_INT(udiStatus2);
				tyNotificationSnd.tyData.sDescription		:= a_tyAlmText[udiStatus2].sAlmText;

			END_IF
		END_IF

		IF tyMsgTypeRcv.bStopTransport = TRUE THEN
			udiStatus2	:= fHermesChkParamSOT(tyStopTransport);

			IF udiStatus2 <> 0 THEN
				eStatus2	:= Error;

				IF udiStatus2 = 2742 THEN
					udiStatus2	:= 10099;	//TransferState Missing While Checking Stop Transport
				ELSIF udiStatus2 = 2743 THEN
					udiStatus2	:= 10100;	//BoardId Missing While Checking Stop Transport
				END_IF

				fHermesAddOneMsgSend(ADR(a_eMsgSend) , ADR(udiMsgSendBffr) , HermesMsgTypeNotification);

				tyNotificationSnd.tyAvl.bSeverity			:= TRUE;
				tyNotificationSnd.tyAvl.bNotificationCode	:= TRUE;
				tyNotificationSnd.tyAvl.bDescription		:= TRUE;
				tyNotificationSnd.tyData.eSeverity			:= HermesSeverityError;
				tyNotificationSnd.tyData.iNotificationCode	:= UDINT_TO_INT(udiStatus2);
				tyNotificationSnd.tyData.sDescription		:= a_tyAlmText[udiStatus2].sAlmText;

			END_IF
		END_IF

		IF tyServiceDescriptionRcv.tyAvl.tySupportedFeatures.bFeatureQueryBoardInfo = TRUE AND p_tyParam.bFeatureSendBoardInfo THEN
			IF tyMsgTypeRcv.bQueryBoardInfo = TRUE THEN
				udiStatus2	:= fHermesChkParamQBI(tyQueryBoardInfo);

				IF udiStatus2 <> 0 THEN
					eStatus2	:= Error;

					IF udiStatus2 = 2766 THEN
						udiStatus2	:= 10102;	//Barcode Missing While Checking Query Board Info
					END_IF

					fHermesAddOneMsgSend(ADR(a_eMsgSend) , ADR(udiMsgSendBffr) , HermesMsgTypeNotification);

					tyNotificationSnd.tyAvl.bSeverity			:= TRUE;
					tyNotificationSnd.tyAvl.bNotificationCode	:= TRUE;
					tyNotificationSnd.tyAvl.bDescription		:= TRUE;
					tyNotificationSnd.tyData.eSeverity			:= HermesSeverityError;
					tyNotificationSnd.tyData.iNotificationCode	:= UDINT_TO_INT(udiStatus2);
					tyNotificationSnd.tyData.sDescription		:= a_tyAlmText[udiStatus2].sAlmText;

		        	tyMsgTypeRcv.bQueryBoardInfo := FALSE; //reset, else will latching
				END_IF
			END_IF
		END_IF

    END_IF

END_ACTION
```

#### Act_Background_ProcessData.st
```iecst
(** 2021-08-01 **)
ACTION Act_Background_ProcessData:

	//Pass Board Available data and TransportFinished BOOL to "BoardDeparted" (SupervisoryHermes)

	tyBoardDepartedInfo := tyBoardAvailableSnd;

	IF EDGEPOS (fbSequenceDS.eMsgTypeSnd = HermesMsgTypeTransportFinished) THEN
		bTransportFinishedSnd := TRUE;
	END_IF

	//Auto Reset bTransportFinishedSnd
	fbSendTm(IN := bTransportFinishedSnd, PT := T#0.3S);
	IF fbSendTm.Q = TRUE THEN
		fbSendTm(IN := FALSE);

		bTransportFinishedSnd	:= FALSE;
	END_IF

	//For Power On or Transfer New Program, udiBAIndex will reset to 0. To find which array sBoardId is empty and continue writing.
	IF udiBAIndex = 0 AND p_bLinkStartupRun = FALSE THEN

		udiTargetAddress := ADR(a_tyBoardDepartedInfo[0].tyData.sBoardId); //Start address
		udiSizeAddress   := SIZEOF(a_tyBoardDepartedInfo[0]); //Size of one array

		FOR i := 0 TO 49 DO //50 Boards Data

			IF memcmp((udiTargetAddress)+(i*udiSizeAddress), ADR('') , 1) = 0 THEN

				bFoundIndex	:= TRUE;
				udiBAIndex := i;
				EXIT;
			END_IF

		END_FOR
	END_IF

	//Retain last 50 PCB handled Boards Data
	p_udiRetainDataAddr	:= ADR(a_tyBoardDepartedInfo);
	p_udiRetainDataLen	:= SIZEOF(a_tyBoardDepartedInfo);

	//Write BoardAvailable Data into arrays and store after send out TransportFinished
	IF EDGENEG(bTransportFinishedSnd) THEN

		memset(ADR(a_tyBoardDepartedInfo[udiBAIndex]) , 0 , SIZEOF(a_tyBoardDepartedInfo[udiBAIndex]));
		memcpy(ADR(a_tyBoardDepartedInfo[udiBAIndex]) , ADR(tyBoardDepartedInfo) , SIZEOF(tyBoardDepartedInfo));

		udiBAIndex	:= udiBAIndex + 1;

		p_eAct := HermesActWriteRetain;

	END_IF

	IF eStatus = Done AND eStat = HermesActWriteRetain THEN
		p_eAct		:= HermesActIdle;
	END_IF

	IF udiBAIndex >= 50 THEN
	   udiBAIndex := 0;
	END_IF

	//BoardForecast
	bFeatureBoardForecast := (p_tyParam.bFeatureBoardForecast = TRUE) AND (tyServiceDescriptionRcv.tyAvl.tySupportedFeatures.bFeatureBoardForecast = TRUE) (*AND bHandshakeDone*) ;

	//New Product can come anytime from Upstream / Select From Product Setting
	IF EDGEPOS (p_bNewProduct) THEN //p_bNewProduct will be True only when machine accepted new recipe, can perform ChangeOver, i.e Machine Free (all zones).
		bNewChangeOver := TRUE;
		idxBoardForecastId	:= 0;//index to send B.F(Id)
	END_IF

	//New Width
	IF EDGEPOS (p_bNewWidth) THEN //p_bSiemensNewProduct will be True only when machine accepted new recipe, can perform ChangeOver, i.e Machine Free (all zones).
		bNewChangeOver := TRUE;
		idxBoardForecastId	:= 0;//index to send B.F(Id)
	END_IF

	IF bFeatureBoardForecast = TRUE THEN
		fbSendBFRstTmr;
		IF bNewChangeOver AND bAllZonesEmpty AND p_bInitDone THEN //Machine Free (all zones)
			bSendBFId := TRUE;
			bNewChangeOver := FALSE;
			fbSendBFRstTmr(IN:= TRUE);
		ELSIF fbSendBFRstTmr.Q THEN
			fbSendBFRstTmr(IN:= FALSE);
			bSendBFId := FALSE;
		END_IF
	ELSE
		bNewChangeOver := FALSE;
		bSendBFId := FALSE;
		bRstSendBFId := FALSE;
		idxBoardForecastId	    := 0;
		idxBoardForecastNoId	:= 0;
	END_IF

	//Reset bSendBFId and idxBoardForecastId	after receive Machine Ready(Id) or Machine Ready()
	IF bRstSendBFId THEN
		bSendBFId := FALSE;
		bRstSendBFId := FALSE;
		idxBoardForecastId	:= 0;
	END_IF

//	//Reset both idxBoardForecastId under handshake condition. Note: idxBoardForecastId only send once.
//	IF (fbSequenceDS.eState <> HermesStateNotAvailableNotReady) AND (fbSequenceDS.eState <> HermesStateMachineReady) AND (fbSequenceDS.eState <> HermesStateBoardAvailable) AND (fbSequenceDS.eState <> HermesStateAvailableAndReady) AND bHandshakeDone = TRUE THEN
//		idxBoardForecastId	:= 0;//index to send B.F(Id)
//	END_IF

	//Reset idxBoardForecastNoId when incoming zone empty
	IF p_bFirstZoneHaveBoard =FALSE AND p_bFirstZoneEndSen = FALSE THEN
		idxBoardForecastNoId	:= 0;//index to send B.F()
	END_IF

END_ACTION
```

#### Act_Background_Sequence.st
```iecst
 (** 2021-08-01 **)
ACTION Act_Background_Sequence:

	IF eStatus1 <> Error THEN

		IF p_bOpsRun = FALSE THEN
			p_bSndIncompl	:= TRUE;
		END_IF

		IF tyMsgTypeRcv.bStopTransport = TRUE THEN
			IF tyStopTransport.tyData.eTransferState = HermesTransferStateNotStarted THEN
				p_bSndNotStart	:= TRUE;
			ELSIF tyStopTransport.tyData.eTransferState = HermesTransferStateIncomplete THEN
				p_bSndIncompl	:= TRUE;
			END_IF
		END_IF

		//Sequence
		fbSequenceDS.bRstState		        := bRstState;
		fbSequenceDS.bRdySnd	        	:= p_bRdySnd; //Machine in OpsG step DSCommTmr (Have DBA)
		fbSequenceDS.bSndCompl	        	:= p_bSndCompl; //Send TransportFinished Msg = Complete (Value = 3)
		fbSequenceDS.bSndIncompl        	:= p_bSndIncompl; //Send TransportFinished Msg = Incomplete (Value = 2)
		fbSequenceDS.bSndNotStart        	:= p_bSndNotStart; //Send TransportFinished Msg = Not Started (Value = 1)
		fbSequenceDS.bFeatureBoardForecast	:= bFeatureBoardForecast; //Feature BoardForecast
		fbSequenceDS.bOpsRun	        	:= p_bOpsRun; //Machine in AutoMode
		fbSequenceDS.bSendBFId              := bSendBFId; //Send B.F with forecast ID, then block Hermes.eState until Downstream reply a MachineReady(Id) or MachineReady()
		fbSequenceDS.bFirstZoneHaveBoard	:= p_bFirstZoneHaveBoard; //First Zone Have Board
		fbSequenceDS.bFirstZoneEndSen	    := p_bFirstZoneEndSen; //First Zone End sensor
		fbSequenceDS.bAllZonesEmpty	        := bAllZonesEmpty; //All Zones empty
		fbSequenceDS(bEn := TRUE);
		bUSRdy		                       	:= fbSequenceDS.bUSRdy;
		bDSRdy			                    := fbSequenceDS.bDSRdy;
		bTransporting                      	:= fbSequenceDS.bTransporting;
		bStopTransport                     	:= fbSequenceDS.bStopTransport;

		IF EDGEPOS(tyMsgTypeRcv.bMachineReady = TRUE) THEN
			bRstSendBFId := TRUE;
		END_IF

		bUSGdRdy	:= (tyBoardAvailableSnd.tyAvl.bFailedBoard = FALSE) OR ((tyBoardAvailableSnd.tyAvl.bFailedBoard = TRUE) AND (tyBoardAvailableSnd.tyData.eFailedBoard <> HermesFailedBoard));

		bDSGdRdy	:= (tyMachineReady.tyAvl.bFailedBoard = FALSE) OR ((tyMachineReady.tyAvl.bFailedBoard = TRUE) AND (tyMachineReady.tyData.eFailedBoard <> HermesFailedBoard));

		IF fbSequenceDS.eState >= HermesStateNotAvailableNotReady THEN
			bHandshakeDone	:= TRUE;
		ELSE
			bHandshakeDone	:= FALSE;
		END_IF

		IF EDGEPOS(fbSequenceDS.eState = HermesStateTransporting) THEN
			p_bSndCompl		:= FALSE;
			p_bSndIncompl	:= FALSE;
			p_bSndNotStart	:= FALSE;
		END_IF

		IF fbSequenceDS.eMsgTypeSnd = HermesMsgTypeServiceDescription THEN
			fHermesAddOneMsgSend(ADR(a_eMsgSend) , ADR(udiMsgSendBffr) , HermesMsgTypeServiceDescription);

			tyServiceDescriptionSnd.tyData.sMachineId								    	:= p_sMcId;
			tyServiceDescriptionSnd.tyData.iLaneId											:= p_tyParam.iLaneID;
			tyServiceDescriptionSnd.tyData.sInterfaceId										:= p_tyParam.sDownstreamInterfaceId;
			tyServiceDescriptionSnd.tyData.sVersion											:= p_sVersion;
			tyServiceDescriptionSnd.tyData.tySupportedFeatures.bFeatureCheckAliveResponse	:= (p_tyParam.bFeatureCheckAliveResponse) AND (p_tyParam.tRcvAlive <> T#0s) AND (p_tyParam.tSndAlive <> T#0s);
			tyServiceDescriptionSnd.tyData.tySupportedFeatures.bFeatureBoardForecast		:= p_tyParam.bFeatureBoardForecast;
			tyServiceDescriptionSnd.tyData.tySupportedFeatures.bFeatureQueryBoardInfo		:= FALSE;
			tyServiceDescriptionSnd.tyData.tySupportedFeatures.bFeatureSendBoardInfo		:= p_tyParam.bFeatureSendBoardInfo;
			tyServiceDescriptionSnd.tyAvl.bMachineId										:= tyServiceDescriptionSnd.tyData.sMachineId <> '';
			tyServiceDescriptionSnd.tyAvl.bLaneId											:= tyServiceDescriptionSnd.tyData.iLaneId<>0;
			tyServiceDescriptionSnd.tyAvl.bInterfaceId										:= tyServiceDescriptionSnd.tyData.sInterfaceId <> '';
			tyServiceDescriptionSnd.tyAvl.bVersion											:= TRUE;
			tyServiceDescriptionSnd.tyAvl.bSupportedFeatures								:= p_tyParam.bFeatureCheckAliveResponse OR p_tyParam.bFeatureBoardForecast OR p_tyParam.bFeatureSendBoardInfo;
			tyServiceDescriptionSnd.tyAvl.tySupportedFeatures.bFeatureCheckAliveResponse	:= (p_tyParam.bFeatureCheckAliveResponse) AND (p_tyParam.tRcvAlive <> T#0s) AND (p_tyParam.tSndAlive <> T#0s);
			tyServiceDescriptionSnd.tyAvl.tySupportedFeatures.bFeatureBoardForecast			:= p_tyParam.bFeatureBoardForecast;
			tyServiceDescriptionSnd.tyAvl.tySupportedFeatures.bFeatureQueryBoardInfo		:= FALSE;
			tyServiceDescriptionSnd.tyAvl.tySupportedFeatures.bFeatureSendBoardInfo			:= p_tyParam.bFeatureSendBoardInfo;

		ELSIF fbSequenceDS.eMsgTypeSnd = HermesMsgTypeBoardForecastId THEN //Beside of sProductTypeId, rWidth, other parameters use default. If upstream does not support BoardForecast, then our machine has no data.

			IF p_eLinkCustomerReq = Siemens AND p_sWorkOrderId <> '' THEN

				IF (idxBoardForecastId < 1) THEN

					fHermesAddOneMsgSend(ADR(a_eMsgSend) , ADR(udiMsgSendBffr) , HermesMsgTypeBoardForecast);
					fHermesGenerateUUID(ADR(tyBoardForecastSnd.tyData.sForecastId) , p_tyDTStructure , pa_usiMacAddr); //Generate ForecastID if there is new Product Changeover

					idxBoardForecastId := idxBoardForecastId + 1;

				END_IF

				tyBoardForecastSnd.tyData.rTimeUntilAvailable       := p_rMcCycleTm + p_rAWCycleTm;
				tyBoardForecastSnd.tyData.sBoardId 			        := ''; //p_sHermesBrdId;//''; //no need to send BoardId for HermesMsgTypeBoardForecastId.
				tyBoardForecastSnd.tyData.sBoardIdCreatedBy			:= p_sMcId; //''; //no need to send BoardIdCreatedBy since no BoardId.
				tyBoardForecastSnd.tyData.eFailedBoard				:= p_tyAutoRcpTravLif.eFailedBoard;//p_eFailedBoard;
				tyBoardForecastSnd.tyData.sProductTypeId			:= p_tyAutoRcpTravLif.sProductTypeId;//p_tySendWorkOrderData.tyData.sProductTypeId;
				tyBoardForecastSnd.tyData.eFlippedBoard		    	:= p_tyAutoRcpTravLif.eFlippedBoard;//p_eFlippedBoard;
				tyBoardForecastSnd.tyData.sTopBarcode				:= p_tyAutoRcpTravLif.sTopBarcode;//p_sTopBarcode;
				tyBoardForecastSnd.tyData.sBottomBarcode			:= p_tyAutoRcpTravLif.sBottomBarcode;//p_sBottomBarcode;
				tyBoardForecastSnd.tyData.rLength					:= p_tyAutoRcpTravLif.rLength;//p_tySendWorkOrderData.tyData.rLength;
				tyBoardForecastSnd.tyData.rWidth					:= p_tyAutoRcpTravLif.rWidth;//p_tySendWorkOrderData.tyData.rWidth;
				tyBoardForecastSnd.tyData.rThickness				:= p_tyAutoRcpTravLif.rThickness;//p_tySendWorkOrderData.tyData.rThickness;
				tyBoardForecastSnd.tyData.rConveyorSpeed			:= p_tyAutoRcpTravLif.rConveyorSpeed;//p_rConveyorSpeed; //dont have
				tyBoardForecastSnd.tyData.rTopClearanceHeight		:= p_tyAutoRcpTravLif.rTopClearanceHeight;//p_tySendWorkOrderData.tyData.rTopClearanceHeight;
				tyBoardForecastSnd.tyData.rBottomClearanceHeight	:= p_tyAutoRcpTravLif.rBottomClearanceHeight;//p_tySendWorkOrderData.tyData.rBottomClearanceHeight;
				tyBoardForecastSnd.tyData.rWeight					:= p_tyAutoRcpTravLif.rWeight;//p_tySendWorkOrderData.tyData.rWeight;
				tyBoardForecastSnd.tyData.sWorkOrderId			    := p_tyAutoRcpTravLif.sWorkOrderId;//p_tySendWorkOrderData.tyData.sWorkOrderId;
				tyBoardForecastSnd.tyData.sBatchId		            := p_tyAutoRcpTravLif.sBatchId;//p_tySendWorkOrderData.tyData.sBatchId;

				tyBoardForecastSnd.tyAvl.bForecastId 			    := TRUE;
				tyBoardForecastSnd.tyAvl.bTimeUntilAvailable		:= tyBoardForecastSnd.tyData.rTimeUntilAvailable <> 0;
				tyBoardForecastSnd.tyAvl.bBoardId 				    := tyBoardForecastSnd.tyData.sBoardId <> '';
				tyBoardForecastSnd.tyAvl.bBoardIdCreatedBy 		    := TRUE;
				tyBoardForecastSnd.tyAvl.bFailedBoard 			    := TRUE;
				tyBoardForecastSnd.tyAvl.bProductTypeId 			:= tyBoardForecastSnd.tyData.sProductTypeId <> '';
				tyBoardForecastSnd.tyAvl.bFlippedBoard 			    := TRUE;
				tyBoardForecastSnd.tyAvl.bTopBarcode 			    := tyBoardForecastSnd.tyData.sTopBarcode <> '';
				tyBoardForecastSnd.tyAvl.bBottomBarcode 			:= tyBoardForecastSnd.tyData.sBottomBarcode <> '';
				tyBoardForecastSnd.tyAvl.bLength 				    := tyBoardForecastSnd.tyData.rLength <> 0;
				tyBoardForecastSnd.tyAvl.bWidth 				    := tyBoardForecastSnd.tyData.rWidth <> 0 AND (p_bBFWidthEn = TRUE);
				tyBoardForecastSnd.tyAvl.bThickness 			    := tyBoardForecastSnd.tyData.rThickness <> 0 AND (p_bBFSltEn = TRUE);
				tyBoardForecastSnd.tyAvl.bConveyorSpeed 			:= tyBoardForecastSnd.tyData.rConveyorSpeed <> 0;
				tyBoardForecastSnd.tyAvl.bTopClearanceHeight 		:= tyBoardForecastSnd.tyData.rTopClearanceHeight <> 0 AND (p_bBFSltEn = TRUE);
				tyBoardForecastSnd.tyAvl.bBottomClearanceHeight 	:= tyBoardForecastSnd.tyData.rBottomClearanceHeight <> 0 AND (p_bBFSltEn = TRUE);
				tyBoardForecastSnd.tyAvl.bWeight 			    	:= tyBoardForecastSnd.tyData.rWeight <> 0;
				tyBoardForecastSnd.tyAvl.bWorkOrderId 		    	:= tyBoardForecastSnd.tyData.sWorkOrderId <> '';
				tyBoardForecastSnd.tyAvl.bBatchId 		        	:= tyBoardForecastSnd.tyData.sBatchId <> '';
			ELSE
				IF (idxBoardForecastId < 1) THEN

					fHermesAddOneMsgSend(ADR(a_eMsgSend) , ADR(udiMsgSendBffr) , HermesMsgTypeBoardForecast);
					fHermesGenerateUUID(ADR(tyBoardForecastSnd.tyData.sForecastId) , p_tyDTStructure , pa_usiMacAddr); //Generate ForecastID if there is new Product Changeover

					idxBoardForecastId := idxBoardForecastId + 1;

				END_IF

				tyBoardForecastSnd.tyData.rTimeUntilAvailable       := p_rMcCycleTm + p_rAWCycleTm;
				tyBoardForecastSnd.tyData.sBoardId 			        := ''; //no need to send BoardId for HermesMsgTypeBoardForecastId.
				tyBoardForecastSnd.tyData.sBoardIdCreatedBy			:= ''; //no need to send BoardIdCreatedBy since no BoardId.
				tyBoardForecastSnd.tyData.eFailedBoard 			    := p_eFailedBoard;
				tyBoardForecastSnd.tyData.sProductTypeId 			:= p_sRecipeNm; //recipe0 name = running recipe name
				tyBoardForecastSnd.tyData.eFlippedBoard 			:= p_eFlippedBoard;
				tyBoardForecastSnd.tyData.sTopBarcode 		    	:= p_sTopBarcode;
				tyBoardForecastSnd.tyData.sBottomBarcode 			:= p_sBottomBarcode;
				tyBoardForecastSnd.tyData.rLength 				    := p_rLength;
				tyBoardForecastSnd.tyData.rWidth 			    	:= DINT_TO_REAL(p_diWidthInUM) / 1000; //recipe 0 width	 = running recipe width
				tyBoardForecastSnd.tyData.rThickness 		    	:= p_rThickness;
				tyBoardForecastSnd.tyData.rConveyorSpeed 			:= p_rConveyorSpeed;
				tyBoardForecastSnd.tyData.rTopClearanceHeight 		:= p_rTopClearanceHeight;
				tyBoardForecastSnd.tyData.rBottomClearanceHeight 	:= p_rBottomClearanceHeight;
				tyBoardForecastSnd.tyData.rWeight 			    	:= p_rWeight;
//				tyBoardForecastSnd.tyData.sWorkOrderId 			    := p_sWorkOrderId;
//				tyBoardForecastSnd.tyData.sBatchId 			        := p_sBatchId;
				tyBoardForecastSnd.tyData.sWorkOrderId 			    := '';
				tyBoardForecastSnd.tyData.sBatchId 			        := '';

				tyBoardForecastSnd.tyAvl.bForecastId 			    := TRUE;
				tyBoardForecastSnd.tyAvl.bTimeUntilAvailable		:= tyBoardForecastSnd.tyData.rTimeUntilAvailable <> 0;
				tyBoardForecastSnd.tyAvl.bBoardId 				    := tyBoardForecastSnd.tyData.sBoardId <> '';
				tyBoardForecastSnd.tyAvl.bBoardIdCreatedBy 		    := TRUE;
				tyBoardForecastSnd.tyAvl.bFailedBoard 			    := TRUE;
				tyBoardForecastSnd.tyAvl.bProductTypeId 			:= tyBoardForecastSnd.tyData.sProductTypeId <> '';
				tyBoardForecastSnd.tyAvl.bFlippedBoard 			    := TRUE;
				tyBoardForecastSnd.tyAvl.bTopBarcode 			    := tyBoardForecastSnd.tyData.sTopBarcode <> '';
				tyBoardForecastSnd.tyAvl.bBottomBarcode 			:= tyBoardForecastSnd.tyData.sBottomBarcode <> '';
				tyBoardForecastSnd.tyAvl.bLength 				    := tyBoardForecastSnd.tyData.rLength <> 0;
				tyBoardForecastSnd.tyAvl.bWidth 				    := tyBoardForecastSnd.tyData.rWidth <> 0 AND (p_bBFWidthEn = TRUE);
				tyBoardForecastSnd.tyAvl.bThickness 			    := tyBoardForecastSnd.tyData.rThickness <> 0 AND (p_bBFSltEn = TRUE);
				tyBoardForecastSnd.tyAvl.bConveyorSpeed 			:= tyBoardForecastSnd.tyData.rConveyorSpeed <> 0;
				tyBoardForecastSnd.tyAvl.bTopClearanceHeight 		:= tyBoardForecastSnd.tyData.rTopClearanceHeight <> 0 AND (p_bBFSltEn = TRUE);
				tyBoardForecastSnd.tyAvl.bBottomClearanceHeight 	:= tyBoardForecastSnd.tyData.rBottomClearanceHeight <> 0 AND (p_bBFSltEn = TRUE);
				tyBoardForecastSnd.tyAvl.bWeight 			    	:= tyBoardForecastSnd.tyData.rWeight <> 0;
				tyBoardForecastSnd.tyAvl.bWorkOrderId 		    	:= tyBoardForecastSnd.tyData.sWorkOrderId <> '';
				tyBoardForecastSnd.tyAvl.bBatchId 		        	:= tyBoardForecastSnd.tyData.sBatchId <> '';
			END_IF

		ELSIF fbSequenceDS.eMsgTypeSnd = HermesMsgTypeBoardForecastNoId THEN

			IF p_eLinkCustomerReq = Siemens AND p_sWorkOrderId <> ''  THEN

				IF p_bNewBrdAvlFirstZone THEN //Generate BoardForecast() by our machine for Manual Load Board at First Zone

					IF (idxBoardForecastNoId < 1) THEN

						fHermesAddOneMsgSend(ADR(a_eMsgSend) , ADR(udiMsgSendBffr) , HermesMsgTypeBoardForecast);

						idxBoardForecastNoId := idxBoardForecastNoId + 1;

					END_IF

					tyBoardForecastSnd.tyData.sForecastId		        := ''; //Do not need to generate ForecastID to downstream

					IF idxBoardForecastNoId <= 1 THEN
						tyBoardForecastSnd.tyData.rTimeUntilAvailable	:= p_rMcCycleTm;
						//				ELSIF idxBoardForecastNoId = 2 THEN
						//					tyBoardForecastSnd.tyData.rTimeUntilAvailable	:= p_rMcCycleTm - (p_rMcCycleTm/3); //divide B.F to 3 segments, open up if needed
						//				ELSIF idxBoardForecastNoId = 3 THEN
						//					tyBoardForecastSnd.tyData.rTimeUntilAvailable	:= p_rMcCycleTm - ((p_rMcCycleTm/3)*2);
					END_IF

					//fHermesGenerateUUID(ADR(tyBoardForecastSnd.tyData.sBoardId) , p_tyDTStructure , pa_usiMacAddr);
					tyBoardForecastSnd.tyData.sBoardId					:= p_sHermesBrdId;
                    tyBoardForecastSnd.tyData.sBoardIdCreatedBy			:= p_sMcId; //no need to send BoardIdCreatedBy since no BoardId.
					tyBoardForecastSnd.tyData.eFailedBoard				:= p_tyAutoRcpTravLif.eFailedBoard;//p_eFailedBoard;
					tyBoardForecastSnd.tyData.sProductTypeId			:= p_tyAutoRcpTravLif.sProductTypeId;//p_tySendWorkOrderData.tyData.sProductTypeId;
					tyBoardForecastSnd.tyData.eFlippedBoard		    	:= p_tyAutoRcpTravLif.eFlippedBoard;//p_eFlippedBoard;
					tyBoardForecastSnd.tyData.sTopBarcode				:= p_tyAutoRcpTravLif.sTopBarcode;//p_sTopBarcode;
					tyBoardForecastSnd.tyData.sBottomBarcode			:= p_tyAutoRcpTravLif.sBottomBarcode;//p_sBottomBarcode;
					tyBoardForecastSnd.tyData.rLength					:= p_tyAutoRcpTravLif.rLength;//p_tySendWorkOrderData.tyData.rLength;
					tyBoardForecastSnd.tyData.rWidth					:= p_tyAutoRcpTravLif.rWidth;//p_tySendWorkOrderData.tyData.rWidth;
					tyBoardForecastSnd.tyData.rThickness				:= p_tyAutoRcpTravLif.rThickness;//p_tySendWorkOrderData.tyData.rThickness;
					tyBoardForecastSnd.tyData.rConveyorSpeed			:= p_tyAutoRcpTravLif.rConveyorSpeed;//p_rConveyorSpeed; //dont have
					tyBoardForecastSnd.tyData.rTopClearanceHeight		:= p_tyAutoRcpTravLif.rTopClearanceHeight;//p_tySendWorkOrderData.tyData.rTopClearanceHeight;
					tyBoardForecastSnd.tyData.rBottomClearanceHeight	:= p_tyAutoRcpTravLif.rBottomClearanceHeight;//p_tySendWorkOrderData.tyData.rBottomClearanceHeight;
					tyBoardForecastSnd.tyData.rWeight					:= p_tyAutoRcpTravLif.rWeight;//p_tySendWorkOrderData.tyData.rWeight;
					tyBoardForecastSnd.tyData.sWorkOrderId			    := p_tyAutoRcpTravLif.sWorkOrderId;//p_tySendWorkOrderData.tyData.sWorkOrderId;
					tyBoardForecastSnd.tyData.sBatchId		            := p_tyAutoRcpTravLif.sBatchId;//p_tySendWorkOrderData.tyData.sBatchId;

					tyBoardForecastSnd.tyAvl.bForecastId 			    := tyBoardForecastSnd.tyData.sForecastId <> '';
					tyBoardForecastSnd.tyAvl.bTimeUntilAvailable		:= tyBoardForecastSnd.tyData.rTimeUntilAvailable <> 0;
					tyBoardForecastSnd.tyAvl.bBoardId 				    := tyBoardForecastSnd.tyData.sBoardId <> '';
					tyBoardForecastSnd.tyAvl.bBoardIdCreatedBy 	    	:= tyBoardForecastSnd.tyData.sBoardIdCreatedBy <> '';
					tyBoardForecastSnd.tyAvl.bFailedBoard 			    := TRUE;
					tyBoardForecastSnd.tyAvl.bProductTypeId 			:= tyBoardForecastSnd.tyData.sProductTypeId <> '';
					tyBoardForecastSnd.tyAvl.bFlippedBoard 		    	:= TRUE;
					tyBoardForecastSnd.tyAvl.bTopBarcode 			    := tyBoardForecastSnd.tyData.sTopBarcode <> '';
					tyBoardForecastSnd.tyAvl.bBottomBarcode 			:= tyBoardForecastSnd.tyData.sBottomBarcode <> '';
					tyBoardForecastSnd.tyAvl.bLength 				    := tyBoardForecastSnd.tyData.rLength <> 0;
					tyBoardForecastSnd.tyAvl.bWidth 				    := tyBoardForecastSnd.tyData.rWidth <> 0 AND (p_bBFWidthEn = TRUE);
					tyBoardForecastSnd.tyAvl.bThickness 			    := tyBoardForecastSnd.tyData.rThickness <> 0 AND (p_bBFSltEn = TRUE);
					tyBoardForecastSnd.tyAvl.bConveyorSpeed 			:= tyBoardForecastSnd.tyData.rConveyorSpeed <> 0;
					tyBoardForecastSnd.tyAvl.bTopClearanceHeight 		:= tyBoardForecastSnd.tyData.rTopClearanceHeight <>0 AND (p_bBFSltEn = TRUE);
					tyBoardForecastSnd.tyAvl.bBottomClearanceHeight 	:= tyBoardForecastSnd.tyData.rBottomClearanceHeight <>0 AND (p_bBFSltEn = TRUE);
					tyBoardForecastSnd.tyAvl.bWeight 			    	:= tyBoardForecastSnd.tyData.rWeight <> 0;
					tyBoardForecastSnd.tyAvl.bWorkOrderId 		    	:= tyBoardForecastSnd.tyData.sWorkOrderId <> '';
					tyBoardForecastSnd.tyAvl.bBatchId 		        	:= tyBoardForecastSnd.tyData.sBatchId <> '';

				ELSE //take PCB_In Board data (For PCB Transfer in from upstream)

					IF (idxBoardForecastNoId < 1) THEN

						fHermesAddOneMsgSend(ADR(a_eMsgSend) , ADR(udiMsgSendBffr) , HermesMsgTypeBoardForecast);
						idxBoardForecastNoId := idxBoardForecastNoId + 1;

					END_IF

					tyBoardForecastSnd.tyData.sForecastId		            := ''; //Do not need to generate ForecastID to downstream

					IF idxBoardForecastNoId <= 1 THEN
						tyBoardForecastSnd.tyData.rTimeUntilAvailable	    := p_rMcCycleTm;
						//			    ELSIF idxBoardForecastNoId = 2 THEN
						//					tyBoardForecastSnd.tyData.rTimeUntilAvailable    	:= p_rMcCycleTm - (p_rMcCycleTm/3); //divide B.F to 3 segments, open up if needed
						//				ELSIF idxBoardForecastNoId = 3 THEN
						//					tyBoardForecastSnd.tyData.rTimeUntilAvailable	    := p_rMcCycleTm - ((p_rMcCycleTm/3)*2);
					END_IF

					tyBoardForecastSnd.tyData.sBoardId                  := p_tyUSBoardArrivedData.tyData.sBoardId;
					tyBoardForecastSnd.tyData.sBoardIdCreatedBy         := p_tyUSBoardArrivedData.tyData.sBoardIdCreatedBy;
					tyBoardForecastSnd.tyData.eFailedBoard 		    	:= p_tyUSBoardArrivedData.tyData.eFailedBoard;
					tyBoardForecastSnd.tyData.sProductTypeId 			:= p_tyUSBoardArrivedData.tyData.sProductTypeId;
					tyBoardForecastSnd.tyData.eFlippedBoard 			:= p_tyUSBoardArrivedData.tyData.eFlippedBoard;
					tyBoardForecastSnd.tyData.sTopBarcode 		    	:= p_tyUSBoardArrivedData.tyData.sTopBarcode;
					tyBoardForecastSnd.tyData.sBottomBarcode 			:= p_tyUSBoardArrivedData.tyData.sBottomBarcode;
					tyBoardForecastSnd.tyData.rLength 				    := p_tyUSBoardArrivedData.tyData.rLength;
					tyBoardForecastSnd.tyData.rWidth 			    	:= p_tyUSBoardArrivedData.tyData.rWidth;
					tyBoardForecastSnd.tyData.rThickness 		    	:= p_tyUSBoardArrivedData.tyData.rThickness;
					tyBoardForecastSnd.tyData.rConveyorSpeed 			:= p_tyUSBoardArrivedData.tyData.rConveyorSpeed;
					tyBoardForecastSnd.tyData.rTopClearanceHeight 		:= p_tyUSBoardArrivedData.tyData.rTopClearanceHeight;
					tyBoardForecastSnd.tyData.rBottomClearanceHeight 	:= p_tyUSBoardArrivedData.tyData.rBottomClearanceHeight;
					tyBoardForecastSnd.tyData.rWeight 			    	:= p_tyUSBoardArrivedData.tyData.rWeight;
					tyBoardForecastSnd.tyData.sWorkOrderId 		    	:= p_tyUSBoardArrivedData.tyData.sWorkOrderId;
					tyBoardForecastSnd.tyData.sBatchId 		        	:= p_tyUSBoardArrivedData.tyData.sBatchId;

					tyBoardForecastSnd.tyAvl.bForecastId 			    := tyBoardForecastSnd.tyData.sForecastId <> '';
					tyBoardForecastSnd.tyAvl.bTimeUntilAvailable		:= tyBoardForecastSnd.tyData.rTimeUntilAvailable <> 0;
					tyBoardForecastSnd.tyAvl.bBoardId 				    := tyBoardForecastSnd.tyData.sBoardId <> '';
					tyBoardForecastSnd.tyAvl.bBoardIdCreatedBy 	    	:= tyBoardForecastSnd.tyData.sBoardIdCreatedBy <> '';
					tyBoardForecastSnd.tyAvl.bFailedBoard 			    := TRUE;
					tyBoardForecastSnd.tyAvl.bProductTypeId 			:= tyBoardForecastSnd.tyData.sProductTypeId <> '';
					tyBoardForecastSnd.tyAvl.bFlippedBoard 		    	:= TRUE;
					tyBoardForecastSnd.tyAvl.bTopBarcode 			    := tyBoardForecastSnd.tyData.sTopBarcode <> '';
					tyBoardForecastSnd.tyAvl.bBottomBarcode 			:= tyBoardForecastSnd.tyData.sBottomBarcode <> '';
					tyBoardForecastSnd.tyAvl.bLength 				    := tyBoardForecastSnd.tyData.rLength <> 0;
					tyBoardForecastSnd.tyAvl.bWidth 				    := tyBoardForecastSnd.tyData.rWidth <> 0;
					tyBoardForecastSnd.tyAvl.bThickness 			    := tyBoardForecastSnd.tyData.rThickness <> 0;
					tyBoardForecastSnd.tyAvl.bConveyorSpeed 			:= tyBoardForecastSnd.tyData.rConveyorSpeed <> 0;
					tyBoardForecastSnd.tyAvl.bTopClearanceHeight 		:= tyBoardForecastSnd.tyData.rTopClearanceHeight <> 0;
					tyBoardForecastSnd.tyAvl.bBottomClearanceHeight 	:= tyBoardForecastSnd.tyData.rBottomClearanceHeight <> 0;
					tyBoardForecastSnd.tyAvl.bWeight 			    	:= tyBoardForecastSnd.tyData.rWeight <> 0;
					tyBoardForecastSnd.tyAvl.bWorkOrderId 		    	:= tyBoardForecastSnd.tyData.sWorkOrderId <> '';
					tyBoardForecastSnd.tyAvl.bBatchId 		        	:= tyBoardForecastSnd.tyData.sBatchId <> '';

				END_IF
			ELSE //no siemens

				IF p_bNewBrdAvlFirstZone THEN //Generate BoardForecast() by our machine for Manual Load Board at First Zone

					IF (idxBoardForecastNoId < 1) THEN

						fHermesAddOneMsgSend(ADR(a_eMsgSend) , ADR(udiMsgSendBffr) , HermesMsgTypeBoardForecast);

						idxBoardForecastNoId := idxBoardForecastNoId + 1;

					END_IF

					tyBoardForecastSnd.tyData.sForecastId		        := ''; //Do not need to generate ForecastID to downstream

					IF idxBoardForecastNoId <= 1 THEN
						tyBoardForecastSnd.tyData.rTimeUntilAvailable	:= p_rMcCycleTm;
						//				ELSIF idxBoardForecastNoId = 2 THEN
						//					tyBoardForecastSnd.tyData.rTimeUntilAvailable	:= p_rMcCycleTm - (p_rMcCycleTm/3); //divide B.F to 3 segments, open up if needed
						//				ELSIF idxBoardForecastNoId = 3 THEN
						//					tyBoardForecastSnd.tyData.rTimeUntilAvailable	:= p_rMcCycleTm - ((p_rMcCycleTm/3)*2);
					END_IF

					fHermesGenerateUUID(ADR(tyBoardForecastSnd.tyData.sBoardId) , p_tyDTStructure , pa_usiMacAddr);
					tyBoardForecastSnd.tyData.sBoardIdCreatedBy         := p_sMcId;
					tyBoardForecastSnd.tyData.eFailedBoard 		    	:= p_eFailedBoard;
					tyBoardForecastSnd.tyData.sProductTypeId 			:= p_sRecipeNm;	 //recipe 0 name = running recipe name
					tyBoardForecastSnd.tyData.eFlippedBoard 			:= p_eFlippedBoard;
					tyBoardForecastSnd.tyData.sTopBarcode 		    	:= p_sTopBarcode;
					tyBoardForecastSnd.tyData.sBottomBarcode 			:= p_sBottomBarcode;
					tyBoardForecastSnd.tyData.rLength 				    := p_rLength;
					tyBoardForecastSnd.tyData.rWidth 			    	:= DINT_TO_REAL(p_diWidthInUM) / 1000;	//recipe 0 width = running recipe width
					tyBoardForecastSnd.tyData.rThickness 		    	:= p_rThickness;
					tyBoardForecastSnd.tyData.rConveyorSpeed 			:= p_rConveyorSpeed;
					tyBoardForecastSnd.tyData.rTopClearanceHeight 		:= p_rTopClearanceHeight;
					tyBoardForecastSnd.tyData.rBottomClearanceHeight 	:= p_rBottomClearanceHeight;
					tyBoardForecastSnd.tyData.rWeight 			    	:= p_rWeight;
//					tyBoardForecastSnd.tyData.sWorkOrderId 		    	:= p_sWorkOrderId;
//					tyBoardForecastSnd.tyData.sBatchId	    	    	:= p_sBatchId;
					tyBoardForecastSnd.tyData.sWorkOrderId 		    	:= '';
					tyBoardForecastSnd.tyData.sBatchId	    	    	:= '';

					tyBoardForecastSnd.tyAvl.bForecastId 			    := tyBoardForecastSnd.tyData.sForecastId <> '';
					tyBoardForecastSnd.tyAvl.bTimeUntilAvailable		:= tyBoardForecastSnd.tyData.rTimeUntilAvailable <> 0;
					tyBoardForecastSnd.tyAvl.bBoardId 				    := tyBoardForecastSnd.tyData.sBoardId <> '';
					tyBoardForecastSnd.tyAvl.bBoardIdCreatedBy 	    	:= tyBoardForecastSnd.tyData.sBoardIdCreatedBy <> '';
					tyBoardForecastSnd.tyAvl.bFailedBoard 			    := TRUE;
					tyBoardForecastSnd.tyAvl.bProductTypeId 			:= tyBoardForecastSnd.tyData.sProductTypeId <> '';
					tyBoardForecastSnd.tyAvl.bFlippedBoard 		    	:= TRUE;
					tyBoardForecastSnd.tyAvl.bTopBarcode 			    := tyBoardForecastSnd.tyData.sTopBarcode <> '';
					tyBoardForecastSnd.tyAvl.bBottomBarcode 			:= tyBoardForecastSnd.tyData.sBottomBarcode <> '';
					tyBoardForecastSnd.tyAvl.bLength 				    := tyBoardForecastSnd.tyData.rLength <> 0;
					tyBoardForecastSnd.tyAvl.bWidth 				    := tyBoardForecastSnd.tyData.rWidth <> 0 AND (p_bBFWidthEn = TRUE);
					tyBoardForecastSnd.tyAvl.bThickness 			    := tyBoardForecastSnd.tyData.rThickness <> 0 AND (p_bBFSltEn = TRUE);
					tyBoardForecastSnd.tyAvl.bConveyorSpeed 			:= tyBoardForecastSnd.tyData.rConveyorSpeed <> 0;
					tyBoardForecastSnd.tyAvl.bTopClearanceHeight 		:= tyBoardForecastSnd.tyData.rTopClearanceHeight <>0 AND (p_bBFSltEn = TRUE);
					tyBoardForecastSnd.tyAvl.bBottomClearanceHeight 	:= tyBoardForecastSnd.tyData.rBottomClearanceHeight <>0 AND (p_bBFSltEn = TRUE);
					tyBoardForecastSnd.tyAvl.bWeight 			    	:= tyBoardForecastSnd.tyData.rWeight <> 0;
					tyBoardForecastSnd.tyAvl.bWorkOrderId 		    	:= tyBoardForecastSnd.tyData.sWorkOrderId <> '';
					tyBoardForecastSnd.tyAvl.bBatchId 		        	:= tyBoardForecastSnd.tyData.sBatchId <> '';

				ELSE //take PCB_In Board data (For PCB Transfer in from upstream)

					IF (idxBoardForecastNoId < 1) THEN

						fHermesAddOneMsgSend(ADR(a_eMsgSend) , ADR(udiMsgSendBffr) , HermesMsgTypeBoardForecast);
						idxBoardForecastNoId := idxBoardForecastNoId + 1;

					END_IF

					tyBoardForecastSnd.tyData.sForecastId		            := ''; //Do not need to generate ForecastID to downstream

					IF idxBoardForecastNoId <= 1 THEN
						tyBoardForecastSnd.tyData.rTimeUntilAvailable	    := p_rMcCycleTm;
						//			    ELSIF idxBoardForecastNoId = 2 THEN
						//					tyBoardForecastSnd.tyData.rTimeUntilAvailable    	:= p_rMcCycleTm - (p_rMcCycleTm/3); //divide B.F to 3 segments, open up if needed
						//				ELSIF idxBoardForecastNoId = 3 THEN
						//					tyBoardForecastSnd.tyData.rTimeUntilAvailable	    := p_rMcCycleTm - ((p_rMcCycleTm/3)*2);
					END_IF

					tyBoardForecastSnd.tyData.sBoardId                  := p_tyUSBoardArrivedData.tyData.sBoardId;
					tyBoardForecastSnd.tyData.sBoardIdCreatedBy         := p_tyUSBoardArrivedData.tyData.sBoardIdCreatedBy;
					tyBoardForecastSnd.tyData.eFailedBoard 		    	:= p_tyUSBoardArrivedData.tyData.eFailedBoard;
					tyBoardForecastSnd.tyData.sProductTypeId 			:= p_tyUSBoardArrivedData.tyData.sProductTypeId;
					tyBoardForecastSnd.tyData.eFlippedBoard 			:= p_tyUSBoardArrivedData.tyData.eFlippedBoard;
					tyBoardForecastSnd.tyData.sTopBarcode 		    	:= p_tyUSBoardArrivedData.tyData.sTopBarcode;
					tyBoardForecastSnd.tyData.sBottomBarcode 			:= p_tyUSBoardArrivedData.tyData.sBottomBarcode;
					tyBoardForecastSnd.tyData.rLength 				    := p_tyUSBoardArrivedData.tyData.rLength;
					tyBoardForecastSnd.tyData.rWidth 			    	:= p_tyUSBoardArrivedData.tyData.rWidth;
					tyBoardForecastSnd.tyData.rThickness 		    	:= p_tyUSBoardArrivedData.tyData.rThickness;
					tyBoardForecastSnd.tyData.rConveyorSpeed 			:= p_tyUSBoardArrivedData.tyData.rConveyorSpeed;
					tyBoardForecastSnd.tyData.rTopClearanceHeight 		:= p_tyUSBoardArrivedData.tyData.rTopClearanceHeight;
					tyBoardForecastSnd.tyData.rBottomClearanceHeight 	:= p_tyUSBoardArrivedData.tyData.rBottomClearanceHeight;
					tyBoardForecastSnd.tyData.rWeight 			    	:= p_tyUSBoardArrivedData.tyData.rWeight;
					tyBoardForecastSnd.tyData.sWorkOrderId 		    	:= p_tyUSBoardArrivedData.tyData.sWorkOrderId;
					tyBoardForecastSnd.tyData.sBatchId 		        	:= p_tyUSBoardArrivedData.tyData.sBatchId;

					tyBoardForecastSnd.tyAvl.bForecastId 			    := tyBoardForecastSnd.tyData.sForecastId <> '';
					tyBoardForecastSnd.tyAvl.bTimeUntilAvailable		:= tyBoardForecastSnd.tyData.rTimeUntilAvailable <> 0;
					tyBoardForecastSnd.tyAvl.bBoardId 				    := tyBoardForecastSnd.tyData.sBoardId <> '';
					tyBoardForecastSnd.tyAvl.bBoardIdCreatedBy 	    	:= tyBoardForecastSnd.tyData.sBoardIdCreatedBy <> '';
					tyBoardForecastSnd.tyAvl.bFailedBoard 			    := TRUE;
					tyBoardForecastSnd.tyAvl.bProductTypeId 			:= tyBoardForecastSnd.tyData.sProductTypeId <> '';
					tyBoardForecastSnd.tyAvl.bFlippedBoard 		    	:= TRUE;
					tyBoardForecastSnd.tyAvl.bTopBarcode 			    := tyBoardForecastSnd.tyData.sTopBarcode <> '';
					tyBoardForecastSnd.tyAvl.bBottomBarcode 			:= tyBoardForecastSnd.tyData.sBottomBarcode <> '';
					tyBoardForecastSnd.tyAvl.bLength 				    := tyBoardForecastSnd.tyData.rLength <> 0;
					tyBoardForecastSnd.tyAvl.bWidth 				    := tyBoardForecastSnd.tyData.rWidth <> 0;
					tyBoardForecastSnd.tyAvl.bThickness 			    := tyBoardForecastSnd.tyData.rThickness <> 0;
					tyBoardForecastSnd.tyAvl.bConveyorSpeed 			:= tyBoardForecastSnd.tyData.rConveyorSpeed <> 0;
					tyBoardForecastSnd.tyAvl.bTopClearanceHeight 		:= tyBoardForecastSnd.tyData.rTopClearanceHeight <> 0;
					tyBoardForecastSnd.tyAvl.bBottomClearanceHeight 	:= tyBoardForecastSnd.tyData.rBottomClearanceHeight <> 0;
					tyBoardForecastSnd.tyAvl.bWeight 			    	:= tyBoardForecastSnd.tyData.rWeight <> 0;
					tyBoardForecastSnd.tyAvl.bWorkOrderId 		    	:= tyBoardForecastSnd.tyData.sWorkOrderId <> '';
					tyBoardForecastSnd.tyAvl.bBatchId 		        	:= tyBoardForecastSnd.tyData.sBatchId <> '';

				END_IF
			END_IF

		ELSIF fbSequenceDS.eMsgTypeSnd = HermesMsgTypeBoardAvailable THEN
			fHermesAddOneMsgSend(ADR(a_eMsgSend) , ADR(udiMsgSendBffr) , HermesMsgTypeBoardAvailable);

				IF (p_eLinkCustomerReq = NA OR p_sWorkOrderId = '') (*OR p_usiProdRcpCurrRcp1McMod = 0)*) AND p_bNewBrdAvlLastZone = TRUE AND p_bRcvBoardInfo = FALSE THEN //Generate New B.A for Unknown PCB

					fHermesGenerateUUID(ADR(tyBoardAvailableSnd.tyData.sBoardId) , p_tyDTStructure , pa_usiMacAddr);

					tyBoardAvailableSnd.tyData.sBoardIdCreatedBy        := p_sMcId; //Generate by our Machine
					tyBoardAvailableSnd.tyData.eFailedBoard				:= p_eFailedBoard;
					tyBoardAvailableSnd.tyData.sProductTypeId			:= p_sRecipeNm;
					tyBoardAvailableSnd.tyData.eFlippedBoard			:= p_eFlippedBoard;
					tyBoardAvailableSnd.tyData.sTopBarcode				:= p_sTopBarcode;
					tyBoardAvailableSnd.tyData.sBottomBarcode			:= p_sBottomBarcode;
					tyBoardAvailableSnd.tyData.rLength					:= p_rLength;
					tyBoardAvailableSnd.tyData.rWidth					:= DINT_TO_REAL(p_diWidthInUM) / 1000;
					tyBoardAvailableSnd.tyData.rThickness				:= p_rThickness;
					tyBoardAvailableSnd.tyData.rConveyorSpeed			:= p_rConveyorSpeed;
					tyBoardAvailableSnd.tyData.rTopClearanceHeight		:= p_rTopClearanceHeight;
					tyBoardAvailableSnd.tyData.rBottomClearanceHeight	:= p_rBottomClearanceHeight;
					tyBoardAvailableSnd.tyData.rWeight					:= p_rWeight;
//					tyBoardAvailableSnd.tyData.sWorkOrderId			    := p_sWorkOrderId;
//					tyBoardAvailableSnd.tyData.sBatchId			        := p_sBatchId;
					tyBoardAvailableSnd.tyData.sWorkOrderId			    := '';
					tyBoardAvailableSnd.tyData.sBatchId			        := '';

					tyBoardAvailableSnd.tyAvl.bBoardId					:= tyBoardAvailableSnd.tyData.sBoardId<>'';
					tyBoardAvailableSnd.tyAvl.bBoardIdCreatedBy			:= tyBoardAvailableSnd.tyData.sBoardIdCreatedBy <> '';
					tyBoardAvailableSnd.tyAvl.bFailedBoard				:= TRUE;
					tyBoardAvailableSnd.tyAvl.bProductTypeId			:= tyBoardAvailableSnd.tyData.sProductTypeId <> '';
					tyBoardAvailableSnd.tyAvl.bFlippedBoard				:= TRUE;
					tyBoardAvailableSnd.tyAvl.bTopBarcode				:= tyBoardAvailableSnd.tyData.sTopBarcode <> '';
					tyBoardAvailableSnd.tyAvl.bBottomBarcode			:= tyBoardAvailableSnd.tyData.sBottomBarcode <> '';
					tyBoardAvailableSnd.tyAvl.bLength					:= tyBoardAvailableSnd.tyData.rLength <> 0;
					tyBoardAvailableSnd.tyAvl.bWidth					:= (tyBoardAvailableSnd.tyData.rWidth <> 0) AND (p_bBAWidthEn = TRUE);
					tyBoardAvailableSnd.tyAvl.bThickness				:= (tyBoardAvailableSnd.tyData.rThickness <> 0) AND (p_bBASltEn = TRUE);
					tyBoardAvailableSnd.tyAvl.bConveyorSpeed			:= tyBoardAvailableSnd.tyData.rConveyorSpeed <> 0;
					tyBoardAvailableSnd.tyAvl.bTopClearanceHeight		:= (tyBoardAvailableSnd.tyData.rTopClearanceHeight <> 0) AND (p_bBASltEn = TRUE);
					tyBoardAvailableSnd.tyAvl.bBottomClearanceHeight	:= (tyBoardAvailableSnd.tyData.rBottomClearanceHeight <> 0) AND (p_bBASltEn = TRUE);
					tyBoardAvailableSnd.tyAvl.bWeight					:= tyBoardAvailableSnd.tyData.rWeight <> 0;
					tyBoardAvailableSnd.tyAvl.bWorkOrderId				:= tyBoardAvailableSnd.tyData.sWorkOrderId <> '';
					tyBoardAvailableSnd.tyAvl.bBatchId			    	:= tyBoardAvailableSnd.tyData.sBatchId <> '';

				ELSIF p_eLinkCustomerReq = Siemens AND p_sWorkOrderId <>'' (*AND (p_usiProdRcpCurrRcp1McMod = 1)*)  AND p_bNewBrdAvlLastZone = TRUE AND p_bRcvBoardInfo = FALSE THEN //Data from Supervisory(Siemens)

					//fHermesGenerateUUID(ADR(tyBoardAvailableSnd.tyData.sBoardId) , p_tyDTStructure , pa_usiMacAddr);
					tyBoardAvailableSnd.tyData.sBoardId 				:= p_sHermesBrdId; //generate for forecast , avail and arrived(supv)

					tyBoardAvailableSnd.tyData.sBoardIdCreatedBy        := p_sMcId;
					tyBoardAvailableSnd.tyData.eFailedBoard				:= p_tyAutoRcpTravLif.eFailedBoard;//p_eFailedBoard;
					tyBoardAvailableSnd.tyData.sProductTypeId			:= p_tyAutoRcpTravLif.sProductTypeId;//p_tySendWorkOrderData.tyData.sProductTypeId;
					tyBoardAvailableSnd.tyData.eFlippedBoard			:= p_tyAutoRcpTravLif.eFlippedBoard;//p_eFlippedBoard;
					tyBoardAvailableSnd.tyData.sTopBarcode				:= p_tyAutoRcpTravLif.sTopBarcode;//p_sTopBarcode;
					tyBoardAvailableSnd.tyData.sBottomBarcode			:= p_tyAutoRcpTravLif.sBottomBarcode;//p_sBottomBarcode;
					tyBoardAvailableSnd.tyData.rLength					:= p_tyAutoRcpTravLif.rLength;//p_tySendWorkOrderData.tyData.rLength;
					tyBoardAvailableSnd.tyData.rWidth					:= p_tyAutoRcpTravLif.rWidth;//p_tySendWorkOrderData.tyData.rWidth;
					tyBoardAvailableSnd.tyData.rThickness				:= p_tyAutoRcpTravLif.rThickness;//p_tySendWorkOrderData.tyData.rThickness;
					tyBoardAvailableSnd.tyData.rConveyorSpeed			:= p_tyAutoRcpTravLif.rConveyorSpeed;//p_rConveyorSpeed; //dont have
					tyBoardAvailableSnd.tyData.rTopClearanceHeight		:= p_tyAutoRcpTravLif.rTopClearanceHeight;//p_tySendWorkOrderData.tyData.rTopClearanceHeight;
					tyBoardAvailableSnd.tyData.rBottomClearanceHeight	:= p_tyAutoRcpTravLif.rBottomClearanceHeight;//p_tySendWorkOrderData.tyData.rBottomClearanceHeight;
					tyBoardAvailableSnd.tyData.rWeight					:= p_tyAutoRcpTravLif.rWeight;//p_tySendWorkOrderData.tyData.rWeight;
					tyBoardAvailableSnd.tyData.sWorkOrderId			    := p_tyAutoRcpTravLif.sWorkOrderId;//p_tySendWorkOrderData.tyData.sWorkOrderId;
					tyBoardAvailableSnd.tyData.sBatchId		            := p_tyAutoRcpTravLif.sBatchId;//p_tySendWorkOrderData.tyData.sBatchId;

					tyBoardAvailableSnd.tyAvl.bBoardId					:= tyBoardAvailableSnd.tyData.sBoardId<>'';
					tyBoardAvailableSnd.tyAvl.bBoardIdCreatedBy			:= tyBoardAvailableSnd.tyData.sBoardIdCreatedBy <> '';
					tyBoardAvailableSnd.tyAvl.bFailedBoard				:= TRUE;
					tyBoardAvailableSnd.tyAvl.bProductTypeId			:= tyBoardAvailableSnd.tyData.sProductTypeId <> '';
					tyBoardAvailableSnd.tyAvl.bFlippedBoard				:= TRUE;
					tyBoardAvailableSnd.tyAvl.bTopBarcode				:= tyBoardAvailableSnd.tyData.sTopBarcode <> '';
					tyBoardAvailableSnd.tyAvl.bBottomBarcode			:= tyBoardAvailableSnd.tyData.sBottomBarcode <> '';
					tyBoardAvailableSnd.tyAvl.bLength					:= tyBoardAvailableSnd.tyData.rLength <> 0;
					tyBoardAvailableSnd.tyAvl.bWidth					:= (tyBoardAvailableSnd.tyData.rWidth <> 0) AND (p_bBAWidthEn = TRUE);
					tyBoardAvailableSnd.tyAvl.bThickness				:= (tyBoardAvailableSnd.tyData.rThickness <> 0) AND (p_bBASltEn = TRUE);
					tyBoardAvailableSnd.tyAvl.bConveyorSpeed			:= tyBoardAvailableSnd.tyData.rConveyorSpeed <> 0;
					tyBoardAvailableSnd.tyAvl.bTopClearanceHeight		:= (tyBoardAvailableSnd.tyData.rTopClearanceHeight <> 0) AND (p_bBASltEn = TRUE);
					tyBoardAvailableSnd.tyAvl.bBottomClearanceHeight	:= (tyBoardAvailableSnd.tyData.rBottomClearanceHeight <> 0) AND (p_bBASltEn = TRUE);
					tyBoardAvailableSnd.tyAvl.bWeight					:= tyBoardAvailableSnd.tyData.rWeight <> 0;
					tyBoardAvailableSnd.tyAvl.bWorkOrderId				:= tyBoardAvailableSnd.tyData.sWorkOrderId <> '';
					tyBoardAvailableSnd.tyAvl.bBatchId			    	:= tyBoardAvailableSnd.tyData.sBatchId <> '';

					/////////////////////////////////////////

				ELSIF p_bNewBrdAvlLastZone = TRUE AND p_bRcvBoardInfo = TRUE THEN //Take BoardInfo From "SendBoardInfo", for Manual Insert PCB

					tyBoardAvailableSnd.tyData.sBoardId                 := p_tyBoardInfoData.tyData.sBoardId;
					tyBoardAvailableSnd.tyData.sBoardIdCreatedBy        := p_tyBoardInfoData.tyData.sBoardIdCreatedBy;
					tyBoardAvailableSnd.tyData.eFailedBoard				:= p_tyBoardInfoData.tyData.eFailedBoard;
					tyBoardAvailableSnd.tyData.sProductTypeId			:= p_tyBoardInfoData.tyData.sProductTypeId;
					tyBoardAvailableSnd.tyData.eFlippedBoard			:= p_tyBoardInfoData.tyData.eFlippedBoard;
					tyBoardAvailableSnd.tyData.sTopBarcode				:= p_tyBoardInfoData.tyData.sTopBarcode;
					tyBoardAvailableSnd.tyData.sBottomBarcode			:= p_tyBoardInfoData.tyData.sBottomBarcode;
					tyBoardAvailableSnd.tyData.rLength					:= p_tyBoardInfoData.tyData.rLength;
					tyBoardAvailableSnd.tyData.rWidth					:= p_tyBoardInfoData.tyData.rWidth;
					tyBoardAvailableSnd.tyData.rThickness				:= p_tyBoardInfoData.tyData.rThickness;
					tyBoardAvailableSnd.tyData.rConveyorSpeed			:= p_rConveyorSpeed; //dont have
					tyBoardAvailableSnd.tyData.rTopClearanceHeight		:= p_tyBoardInfoData.tyData.rTopClearanceHeight;
					tyBoardAvailableSnd.tyData.rBottomClearanceHeight	:= p_tyBoardInfoData.tyData.rBottomClearanceHeight;
					tyBoardAvailableSnd.tyData.rWeight					:= p_tyBoardInfoData.tyData.rWeight;
					tyBoardAvailableSnd.tyData.sWorkOrderId			    := p_tyBoardInfoData.tyData.sWorkOrderId;
					tyBoardAvailableSnd.tyData.sBatchId		            := p_tyBoardInfoData.tyData.sBatchId;

					tyBoardAvailableSnd.tyAvl.bBoardId					:= tyBoardAvailableSnd.tyData.sBoardId <> '';
					tyBoardAvailableSnd.tyAvl.bBoardIdCreatedBy			:= tyBoardAvailableSnd.tyData.sBoardIdCreatedBy <> '';
					tyBoardAvailableSnd.tyAvl.bFailedBoard				:= TRUE;
					tyBoardAvailableSnd.tyAvl.bProductTypeId			:= tyBoardAvailableSnd.tyData.sProductTypeId <> '';
					tyBoardAvailableSnd.tyAvl.bFlippedBoard				:= TRUE;
					tyBoardAvailableSnd.tyAvl.bTopBarcode				:= tyBoardAvailableSnd.tyData.sTopBarcode <> '';
					tyBoardAvailableSnd.tyAvl.bBottomBarcode			:= tyBoardAvailableSnd.tyData.sBottomBarcode <> '';
					tyBoardAvailableSnd.tyAvl.bLength					:= tyBoardAvailableSnd.tyData.rLength <> 0;
					tyBoardAvailableSnd.tyAvl.bWidth					:= (tyBoardAvailableSnd.tyData.rWidth <> 0);
					tyBoardAvailableSnd.tyAvl.bThickness				:= (tyBoardAvailableSnd.tyData.rThickness <> 0);
					tyBoardAvailableSnd.tyAvl.bConveyorSpeed			:= tyBoardAvailableSnd.tyData.rConveyorSpeed <> 0;
					tyBoardAvailableSnd.tyAvl.bTopClearanceHeight		:= (tyBoardAvailableSnd.tyData.rTopClearanceHeight <> 0);
					tyBoardAvailableSnd.tyAvl.bBottomClearanceHeight	:= (tyBoardAvailableSnd.tyData.rBottomClearanceHeight <> 0);
					tyBoardAvailableSnd.tyAvl.bWeight					:= tyBoardAvailableSnd.tyData.rWeight <> 0;
					tyBoardAvailableSnd.tyAvl.bWorkOrderId				:= tyBoardAvailableSnd.tyData.sWorkOrderId <> '';
					tyBoardAvailableSnd.tyAvl.bBatchId			    	:= tyBoardAvailableSnd.tyData.sBatchId <> '';

		ELSE //Take from PCB_In Board Data

			fbParseBrdAvlExternal.p_XMLTable		:= ADR(pa_tyXMLTableDataBrdAvl); //last zone B.A
			fbParseBrdAvlExternal.iTotalIdxWrite	:= p_iXMLTableDataBrdAvlTtlIdx; //last zone
			fbParseBrdAvlExternal;
			tyBoardAvailableSnd	:= fbParseBrdAvlExternal.tyBoardAvailable;
		END_IF

	ELSIF fbSequenceDS.eMsgTypeSnd = HermesMsgTypeRevokeBoardAvl THEN
		fHermesAddOneMsgSend(ADR(a_eMsgSend) , ADR(udiMsgSendBffr) , HermesMsgTypeRevokeBoardAvl);

	ELSIF fbSequenceDS.eMsgTypeSnd = HermesMsgTypeTransportFinished THEN
		fHermesAddOneMsgSend(ADR(a_eMsgSend) , ADR(udiMsgSendBffr) , HermesMsgTypeTransportFinished);

		IF p_bSndCompl = TRUE THEN
			tyTransportFinished.tyData.eTransferState	:= HermesTransferStateComplete;
		ELSIF p_bSndIncompl = TRUE THEN
			tyTransportFinished.tyData.eTransferState	:= HermesTransferStateIncomplete;
		ELSE
			tyTransportFinished.tyData.eTransferState	:= HermesTransferStateNotStarted;
		END_IF
		tyTransportFinished.tyData.sBoardId				:= tyStartTransport.tyData.sBoardId;

		tyTransportFinished.tyAvl.bTransferState		:= TRUE;
		tyTransportFinished.tyAvl.bBoardId				:= TRUE;

	END_IF

	END_IF

END_ACTION
```

#### Act_Background_TCPRcv.st
```iecst
(** 2021-08-01 **)
ACTION Act_Background_TCPRcv:

	IF eStatus1 <> Error THEN

		//Receive Data
		IF p_bInternalUse = FALSE THEN
			fbRcv.udiTCPIdent	:= udiClntIdent;
			fbRcv(bEn := TRUE);
		ELSE
			sRcv	:= p_sInternalRcv;
		END_IF

		IF (fbRcv.udiStatus = 0) OR ((p_bInternalUse = TRUE) AND (LEN(sRcv) > 0)) THEN

			fLogDTConvert(ADR(sDT) , p_dtCurrDT);
			memset(ADR(a_sLogList[udiLogCntr]) , 0 , SIZEOF(a_sLogList[udiLogCntr]));
			memcpy(ADR(a_sLogList[udiLogCntr]) + LEN(a_sLogList[udiLogCntr]) , ADR(sDT) , LEN(sDT));
			memcpy(ADR(a_sLogList[udiLogCntr]) + LEN(a_sLogList[udiLogCntr]) , ADR('$r$n') , LEN('$r$n'));
			memcpy(ADR(a_sLogList[udiLogCntr]) + LEN(a_sLogList[udiLogCntr]) , ADR('RCV_FRM_DS$r$n') , LEN('RCV_FRM_DS$r$n'));
			memcpy(ADR(a_sLogList[udiLogCntr]) + LEN(a_sLogList[udiLogCntr]) , ADR(sRcv) , LEN(sRcv));
			memcpy(ADR(a_sLogList[udiLogCntr]) + LEN(a_sLogList[udiLogCntr]) , ADR('$r$n$r$n') , LEN('$r$n$r$n'));

			udiLogCntr	:= udiLogCntr + 1;
			IF udiLogCntr = 11 THEN
				udiLogCntr	:= 1;
			END_IF

			fXMLConvertToTable(ADR(sRcv) , LEN(sRcv) , ADR(a_tyXMLTableDataRcv) , ADR(a_tyXMLTableDataRcv[0].sTitle) , SIZEOF(a_tyXMLTableDataRcv[0].sTitle) , ADR(a_tyXMLTableDataRcv[0].sValue) , SIZEOF(a_tyXMLTableDataRcv[0].sValue) , ADR(a_tyXMLTableDataRcv[0].uiSize) , SIZEOF(a_tyXMLTableDataRcv[0]) , SIZEOF(a_tyXMLTableDataRcv) / SIZEOF(a_tyXMLTableDataRcv[0]) , ADR(udiXMLTableWriteIdx));

			fbParseXMLTable.iTotalIdxWrite	:= UDINT_TO_INT(udiXMLTableWriteIdx);
			fbParseXMLTable;

			IF fbParseXMLTable.tyMsgType.bCheckAlive = TRUE THEN
				tyMsgTypeRcv.bCheckAlive	:= TRUE;
				tyCheckAliveRcv				:= fbParseXMLTable.tyCheckAlive;
			END_IF

			IF fbParseXMLTable.tyMsgType.bCheckAlivePing = TRUE THEN
				tyMsgTypeRcv.bCheckAlivePing	:= TRUE;
				tyCheckAlivePingRcv				:= fbParseXMLTable.tyCheckAlivePing;
			END_IF

			IF fbParseXMLTable.tyMsgType.bCheckAlivePong = TRUE THEN
				tyMsgTypeRcv.bCheckAlivePong	:= TRUE;
				tyCheckAlivePongRcv				:= fbParseXMLTable.tyCheckAlivePong;
			END_IF

			IF fbParseXMLTable.tyMsgType.bServiceDescription = TRUE THEN
				tyMsgTypeRcv.bServiceDescription	:= TRUE;
				tyServiceDescriptionRcv				:= fbParseXMLTable.tyServiceDescription;
			END_IF

			IF fbParseXMLTable.tyMsgType.bNotification = TRUE THEN
				tyMsgTypeRcv.bNotification	:= TRUE;
				tyNotificationRcv			:= fbParseXMLTable.tyNotification;
			END_IF

			IF fbParseXMLTable.tyMsgType.bBoardAvailable = TRUE THEN
				tyMsgTypeRcv.bBoardAvailable	:= TRUE;
				tyBoardAvailableRcv				:= fbParseXMLTable.tyBoardAvailable;

				memset(ADR(a_tyXMLTableDataBrdAvl) , 0 , SIZEOF(a_tyXMLTableDataBrdAvl));
				memcpy(ADR(a_tyXMLTableDataBrdAvl) , ADR(a_tyXMLTableDataRcv) + (fbParseXMLTable.iBoardAvailableFirstIdx * SIZEOF(a_tyXMLTableDataRcv[0])) , (fbParseXMLTable.iBoardAvailableLastIdx - fbParseXMLTable.iBoardAvailableFirstIdx + 1) * SIZEOF(a_tyXMLTableDataRcv[0]));

			END_IF

			IF fbParseXMLTable.tyMsgType.bRevokeBoardAvailable = TRUE THEN
				tyMsgTypeRcv.bRevokeBoardAvailable	:= TRUE;
			END_IF

			IF fbParseXMLTable.tyMsgType.bMachineReady = TRUE THEN
				tyMsgTypeRcv.bMachineReady	:= TRUE;
				tyMachineReady				:= fbParseXMLTable.tyMachineReady;
			END_IF

			IF fbParseXMLTable.tyMsgType.bRevokeMachineReady = TRUE THEN
				tyMsgTypeRcv.bRevokeMachineReady	:= TRUE;
			END_IF

			IF fbParseXMLTable.tyMsgType.bStartTransport = TRUE THEN
				tyMsgTypeRcv.bStartTransport	:= TRUE;
				tyStartTransport				:= fbParseXMLTable.tyStartTransport;
			END_IF

			IF fbParseXMLTable.tyMsgType.bStopTransport = TRUE THEN
				tyMsgTypeRcv.bStopTransport	:= TRUE;
				tyStopTransport				:= fbParseXMLTable.tyStopTransport;
			END_IF

			IF fbParseXMLTable.tyMsgType.bTransportFinished = TRUE THEN
				tyMsgTypeRcv.bTransportFinished	:= TRUE;
				tyTransportFinished				:= fbParseXMLTable.tyTransportFinished;
			END_IF

			IF fbParseXMLTable.tyMsgType.bSetConfiguration = TRUE THEN
				tyMsgTypeRcv.bSetConfiguration	:= TRUE;
				tySetConfiguration				:= fbParseXMLTable.tySetConfiguration;
			END_IF

			IF fbParseXMLTable.tyMsgType.bGetConfiguration = TRUE THEN
				tyMsgTypeRcv.bGetConfiguration	:= TRUE;
			END_IF

			IF fbParseXMLTable.tyMsgType.bCurrentConfiguration = TRUE THEN
				tyMsgTypeRcv.bCurrentConfiguration	:= TRUE;
				tyCurrentConfiguration				:= fbParseXMLTable.tyCurrentConfiguration;
			END_IF

			IF fbParseXMLTable.tyMsgType.bBoardForecast = TRUE THEN
				tyMsgTypeRcv.bBoardForecast	:= TRUE;
				tyBoardForecastRcv				:= fbParseXMLTable.tyBoardForecast;
			END_IF

			IF fbParseXMLTable.tyMsgType.bQueryBoardInfo = TRUE THEN
				tyMsgTypeRcv.bQueryBoardInfo	:= TRUE;
				tyQueryBoardInfo				:= fbParseXMLTable.tyQueryBoardInfo;
			END_IF

			IF fbParseXMLTable.tyMsgType.bSendBoardInfo = TRUE THEN
				tyMsgTypeRcv.bSendBoardInfo	:= TRUE;
				tySendBoardInfo				:= fbParseXMLTable.tySendBoardInfo;
			END_IF

			fbRcv(bEn := FALSE);

			memset(ADR(sRcv) , 0 , SIZEOF(sRcv));

		ELSIF (fbRcv.udiStatus = 2317) AND (p_bInternalUse = FALSE) THEN
			fbRcv(bEn := FALSE);

			memset(ADR(sRcv) , 0 , SIZEOF(sRcv));

		ELSIF (fbRcv.udiStatus = 2316) AND (p_bInternalUse = FALSE) THEN
			bRstConnection	:= TRUE;

			memset(ADR(sRcv) , 0 , SIZEOF(sRcv));

		ELSIF (fbRcv.udiStatus = 2318) AND (p_bInternalUse = FALSE) THEN
			bRstConnection	:= TRUE;

			memset(ADR(sRcv) , 0 , SIZEOF(sRcv));

		ELSIF (fbRcv.udiStatus < 65534) AND (p_bInternalUse = FALSE) THEN
			eStatus1	:= Error;

			IF fbRcv.udiStatus = 2300 THEN
				udiStatus1	:= 10014;	//Invalid Ident While Receiving Data
			ELSIF fbRcv.udiStatus = 2319 THEN
				udiStatus1	:= 10015;	//TCP Receive Data Error While Receiving Data
			ELSE
				udiStatus1	:= fbRcv.udiStatus;
			END_IF

			memset(ADR(sRcv) , 0 , SIZEOF(sRcv));

		END_IF

	END_IF

END_ACTION
```
